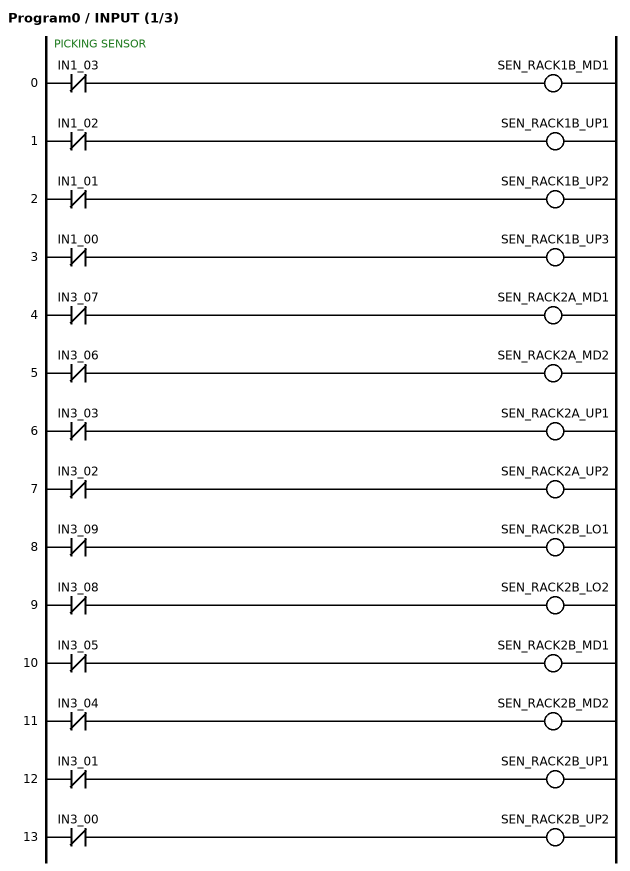
(* [picture p24: Program0 / INPUT, rungs 0-13] *)
(* Rung 0: PICKING SENSOR *)
SEN_RACK1B_MD1 := NOT IN1_03;
(* Rung 1 *)
SEN_RACK1B_UP1 := NOT IN1_02;
(* Rung 2 *)
SEN_RACK1B_UP2 := NOT IN1_01;
(* Rung 3 *)
SEN_RACK1B_UP3 := NOT IN1_00;
(* Rung 4 *)
SEN_RACK2A_MD1 := NOT IN3_07;
(* Rung 5 *)
SEN_RACK2A_MD2 := NOT IN3_06;
(* Rung 6 *)
SEN_RACK2A_UP1 := NOT IN3_03;
(* Rung 7 *)
SEN_RACK2A_UP2 := NOT IN3_02;
(* Rung 8 *)
SEN_RACK2B_LO1 := NOT IN3_09;
(* Rung 9 *)
SEN_RACK2B_LO2 := NOT IN3_08;
(* Rung 10 *)
SEN_RACK2B_MD1 := NOT IN3_05;
(* Rung 11 *)
SEN_RACK2B_MD2 := NOT IN3_04;
(* Rung 12 *)
SEN_RACK2B_UP1 := NOT IN3_01;
(* Rung 13 *)
SEN_RACK2B_UP2 := NOT IN3_00;

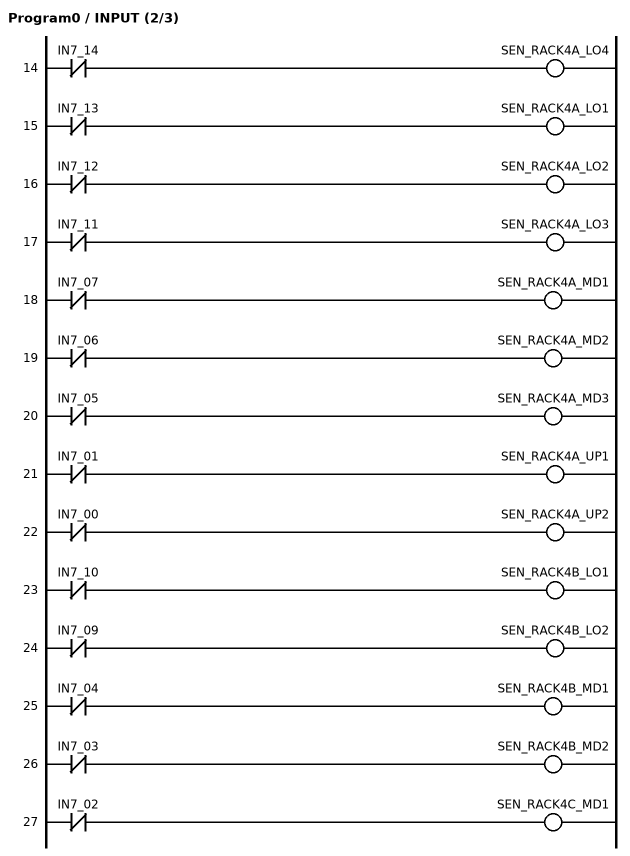
(* Rung 14 *)
SEN_RACK4A_LO4 := NOT IN7_14;
(* Rung 15 *)
SEN_RACK4A_LO1 := NOT IN7_13;
(* Rung 16 *)
SEN_RACK4A_LO2 := NOT IN7_12;
(* Rung 17 *)
SEN_RACK4A_LO3 := NOT IN7_11;
(* Rung 18 *)
SEN_RACK4A_MD1 := NOT IN7_07;
(* Rung 19 *)
SEN_RACK4A_MD2 := NOT IN7_06;
(* Rung 20 *)
SEN_RACK4A_MD3 := NOT IN7_05;
(* Rung 21 *)
SEN_RACK4A_UP1 := NOT IN7_01;
(* Rung 22 *)
SEN_RACK4A_UP2 := NOT IN7_00;
(* Rung 23 *)
SEN_RACK4B_LO1 := NOT IN7_10;
(* Rung 24 *)
SEN_RACK4B_LO2 := NOT IN7_09;
(* Rung 25 *)
SEN_RACK4B_MD1 := NOT IN7_04;
(* Rung 26 *)
SEN_RACK4B_MD2 := NOT IN7_03;
(* Rung 27 *)
SEN_RACK4C_MD1 := NOT IN7_02;

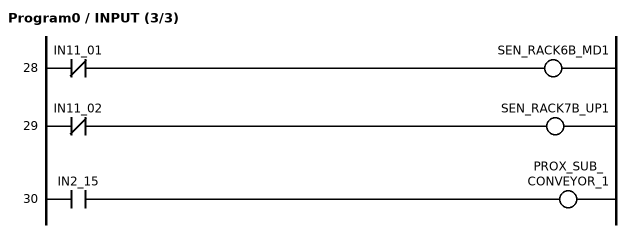
(* Rung 28 *)
SEN_RACK6B_MD1 := NOT IN11_01;
(* Rung 29 *)
SEN_RACK7B_UP1 := NOT IN11_02;
(* Rung 30 *)
PROX_SUB_CONVEYOR_1 := IN2_15;

(* Section OUTPUT: ladder, written here as Structured Text *)

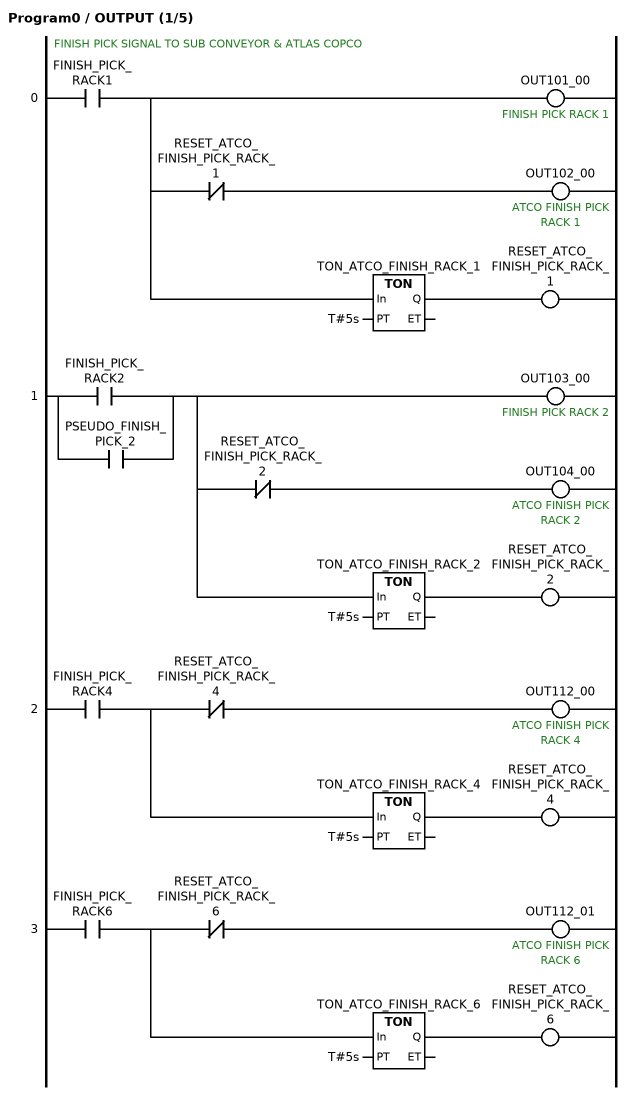
(* Rung 0: FINISH PICK SIGNAL TO SUB CONVEYOR & ATLAS COPCO *)
OUT101_00 := FINISH_PICK_RACK1;
OUT102_00 := FINISH_PICK_RACK1 AND NOT RESET_ATCO_FINISH_PICK_RACK_1;
TON_ATCO_FINISH_RACK_1(In := FINISH_PICK_RACK1, PT := T#5s);
RESET_ATCO_FINISH_PICK_RACK_1 := TON_ATCO_FINISH_RACK_1.Q;
(* Rung 1 *)
OUT103_00 := FINISH_PICK_RACK2 OR PSEUDO_FINISH_PICK_2;
OUT104_00 := (FINISH_PICK_RACK2 OR PSEUDO_FINISH_PICK_2) AND NOT RESET_ATCO_FINISH_PICK_RACK_2;
TON_ATCO_FINISH_RACK_2(In := FINISH_PICK_RACK2 OR PSEUDO_FINISH_PICK_2, PT := T#5s);
RESET_ATCO_FINISH_PICK_RACK_2 := TON_ATCO_FINISH_RACK_2.Q;
(* Rung 2 *)
OUT112_00 := FINISH_PICK_RACK4 AND NOT RESET_ATCO_FINISH_PICK_RACK_4;
TON_ATCO_FINISH_RACK_4(In := FINISH_PICK_RACK4, PT := T#5s);
RESET_ATCO_FINISH_PICK_RACK_4 := TON_ATCO_FINISH_RACK_4.Q;
(* Rung 3 *)
OUT112_01 := FINISH_PICK_RACK6 AND NOT RESET_ATCO_FINISH_PICK_RACK_6;
TON_ATCO_FINISH_RACK_6(In := FINISH_PICK_RACK6, PT := T#5s);
RESET_ATCO_FINISH_PICK_RACK_6 := TON_ATCO_FINISH_RACK_6.Q;

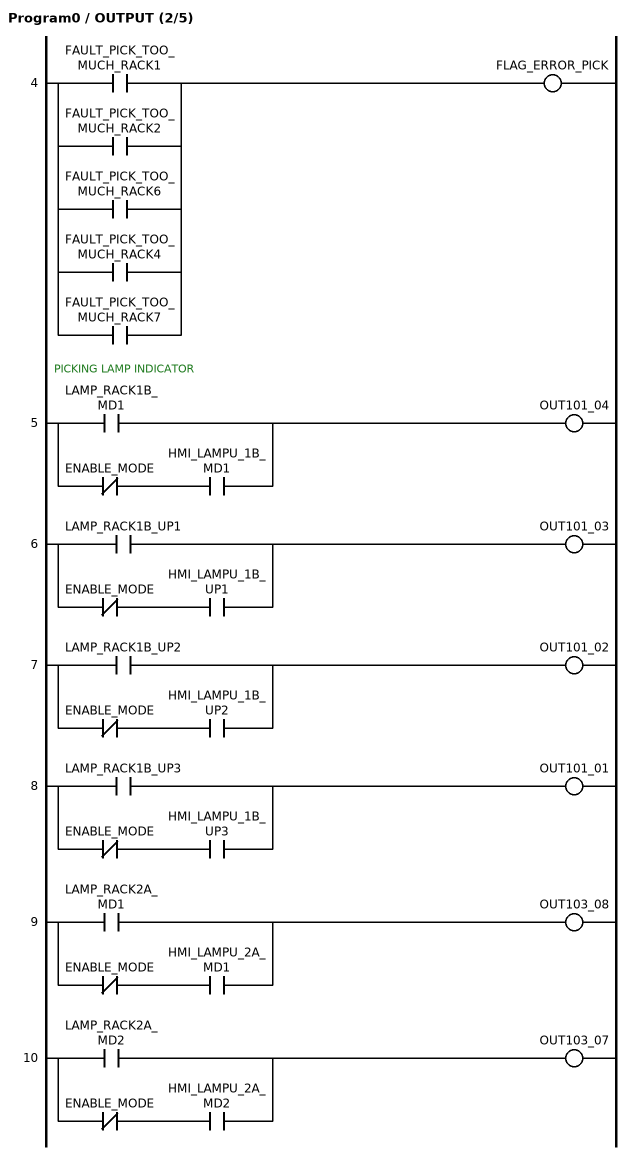
(* Rung 4 *)
FLAG_ERROR_PICK := FAULT_PICK_TOO_MUCH_RACK1 OR FAULT_PICK_TOO_MUCH_RACK2 OR FAULT_PICK_TOO_MUCH_RACK6 OR FAULT_PICK_TOO_MUCH_RACK4 OR FAULT_PICK_TOO_MUCH_RACK7;
(* Rung 5: PICKING LAMP INDICATOR *)
OUT101_04 := LAMP_RACK1B_MD1 OR (NOT ENABLE_MODE AND HMI_LAMPU_1B_MD1);
(* Rung 6 *)
OUT101_03 := LAMP_RACK1B_UP1 OR (NOT ENABLE_MODE AND HMI_LAMPU_1B_UP1);
(* Rung 7 *)
OUT101_02 := LAMP_RACK1B_UP2 OR (NOT ENABLE_MODE AND HMI_LAMPU_1B_UP2);
(* Rung 8 *)
OUT101_01 := LAMP_RACK1B_UP3 OR (NOT ENABLE_MODE AND HMI_LAMPU_1B_UP3);
(* Rung 9 *)
OUT103_08 := LAMP_RACK2A_MD1 OR (NOT ENABLE_MODE AND HMI_LAMPU_2A_MD1);
(* Rung 10 *)
OUT103_07 := LAMP_RACK2A_MD2 OR (NOT ENABLE_MODE AND HMI_LAMPU_2A_MD2);

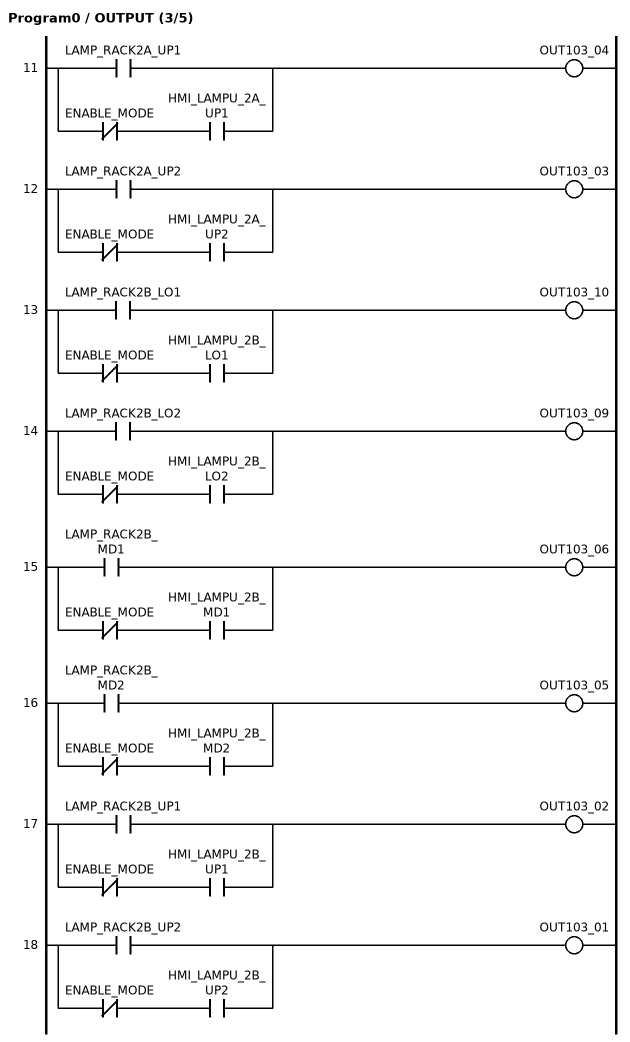
(* Rung 11 *)
OUT103_04 := LAMP_RACK2A_UP1 OR (NOT ENABLE_MODE AND HMI_LAMPU_2A_UP1);
(* Rung 12 *)
OUT103_03 := LAMP_RACK2A_UP2 OR (NOT ENABLE_MODE AND HMI_LAMPU_2A_UP2);
(* Rung 13 *)
OUT103_10 := LAMP_RACK2B_LO1 OR (NOT ENABLE_MODE AND HMI_LAMPU_2B_LO1);
(* Rung 14 *)
OUT103_09 := LAMP_RACK2B_LO2 OR (NOT ENABLE_MODE AND HMI_LAMPU_2B_LO2);
(* Rung 15 *)
OUT103_06 := LAMP_RACK2B_MD1 OR (NOT ENABLE_MODE AND HMI_LAMPU_2B_MD1);
(* Rung 16 *)
OUT103_05 := LAMP_RACK2B_MD2 OR (NOT ENABLE_MODE AND HMI_LAMPU_2B_MD2);
(* Rung 17 *)
OUT103_02 := LAMP_RACK2B_UP1 OR (NOT ENABLE_MODE AND HMI_LAMPU_2B_UP1);
(* Rung 18 *)
OUT103_01 := LAMP_RACK2B_UP2 OR (NOT ENABLE_MODE AND HMI_LAMPU_2B_UP2);

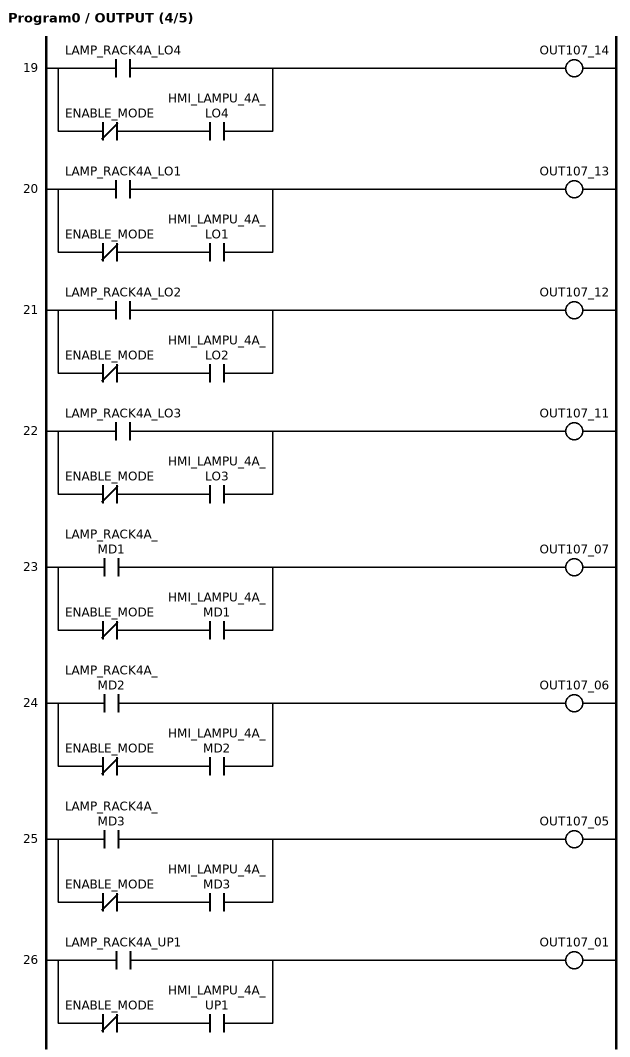
(* Rung 19 *)
OUT107_14 := LAMP_RACK4A_LO4 OR (NOT ENABLE_MODE AND HMI_LAMPU_4A_LO4);
(* Rung 20 *)
OUT107_13 := LAMP_RACK4A_LO1 OR (NOT ENABLE_MODE AND HMI_LAMPU_4A_LO1);
(* Rung 21 *)
OUT107_12 := LAMP_RACK4A_LO2 OR (NOT ENABLE_MODE AND HMI_LAMPU_4A_LO2);
(* Rung 22 *)
OUT107_11 := LAMP_RACK4A_LO3 OR (NOT ENABLE_MODE AND HMI_LAMPU_4A_LO3);
(* Rung 23 *)
OUT107_07 := LAMP_RACK4A_MD1 OR (NOT ENABLE_MODE AND HMI_LAMPU_4A_MD1);
(* Rung 24 *)
OUT107_06 := LAMP_RACK4A_MD2 OR (NOT ENABLE_MODE AND HMI_LAMPU_4A_MD2);
(* Rung 25 *)
OUT107_05 := LAMP_RACK4A_MD3 OR (NOT ENABLE_MODE AND HMI_LAMPU_4A_MD3);
(* Rung 26 *)
OUT107_01 := LAMP_RACK4A_UP1 OR (NOT ENABLE_MODE AND HMI_LAMPU_4A_UP1);

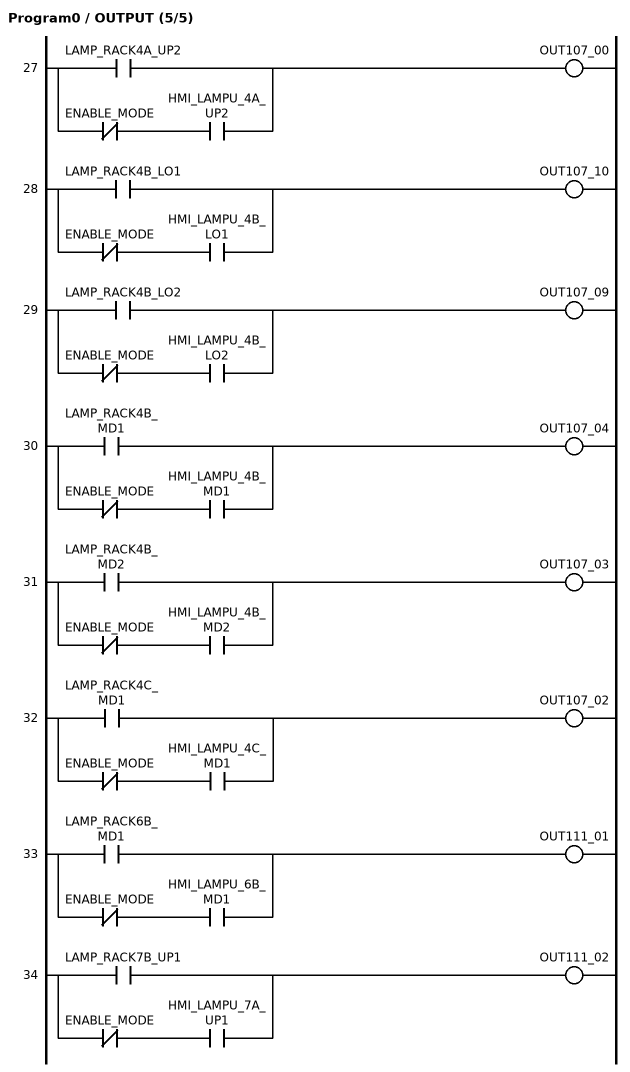
(* Rung 27 *)
OUT107_00 := LAMP_RACK4A_UP2 OR (NOT ENABLE_MODE AND HMI_LAMPU_4A_UP2);
(* Rung 28 *)
OUT107_10 := LAMP_RACK4B_LO1 OR (NOT ENABLE_MODE AND HMI_LAMPU_4B_LO1);
(* Rung 29 *)
OUT107_09 := LAMP_RACK4B_LO2 OR (NOT ENABLE_MODE AND HMI_LAMPU_4B_LO2);
(* Rung 30 *)
OUT107_04 := LAMP_RACK4B_MD1 OR (NOT ENABLE_MODE AND HMI_LAMPU_4B_MD1);
(* Rung 31 *)
OUT107_03 := LAMP_RACK4B_MD2 OR (NOT ENABLE_MODE AND HMI_LAMPU_4B_MD2);
(* Rung 32 *)
OUT107_02 := LAMP_RACK4C_MD1 OR (NOT ENABLE_MODE AND HMI_LAMPU_4C_MD1);
(* Rung 33 *)
OUT111_01 := LAMP_RACK6B_MD1 OR (NOT ENABLE_MODE AND HMI_LAMPU_6B_MD1);
(* Rung 34 *)
OUT111_02 := LAMP_RACK7B_UP1 OR (NOT ENABLE_MODE AND HMI_LAMPU_7A_UP1);
END_PROGRAM

FUNCTION_BLOCK FB_PICKING_SEQ
VAR
    DONE_PICK_1 : BOOL;
    NI_LAMP_PICK_1 : BOOL;
    NI_FAULT_MUCH_LAMP_PICK_1 : BOOL;
    NI_FAULT_FALSE_LAMP_PICK_1 : BOOL;
    DONE_PICK_2 : BOOL;
    NI_LAMP_PICK_2 : BOOL;
    NI_FAULT_MUCH_LAMP_PICK_2 : BOOL;
    NI_FAULT_FALSE_LAMP_PICK_2 : BOOL;
    DONE_PICK_3 : BOOL;
    NI_LAMP_PICK_3 : BOOL;
    NI_FAULT_MUCH_LAMP_PICK_3 : BOOL;
    NI_FAULT_FALSE_LAMP_PICK_3 : BOOL;
    DONE_PICK_4 : BOOL;
    NI_LAMP_PICK_4 : BOOL;
    NI_FAULT_MUCH_LAMP_PICK_4 : BOOL;
    NI_FAULT_FALSE_LAMP_PICK_4 : BOOL;
    DONE_PICK_5 : BOOL;
    NI_LAMP_PICK_5 : BOOL;
    NI_FAULT_MUCH_LAMP_PICK_5 : BOOL;
    NI_FAULT_FALSE_LAMP_PICK_5 : BOOL;
    DONE_PICK_6 : BOOL;
    NI_LAMP_PICK_6 : BOOL;
    NI_FAULT_MUCH_LAMP_PICK_6 : BOOL;
    NI_FAULT_FALSE_LAMP_PICK_6 : BOOL;
    DONE_PICK_7 : BOOL;
    NI_LAMP_PICK_7 : BOOL;
    NI_FAULT_MUCH_LAMP_PICK_7 : BOOL;
    NI_FAULT_FALSE_LAMP_PICK_7 : BOOL;
    NI_LAMP_PICK_8 : BOOL;
    DONE_PICK_8 : BOOL;
    NI_FAULT_MUCH_LAMP_PICK_8 : BOOL;
    NI_FAULT_FALSE_LAMP_PICK_8 : BOOL;
    DONE_PICK_9 : BOOL;
    NI_LAMP_PICK_9 : BOOL;
    NI_FAULT_MUCH_LAMP_PICK_9 : BOOL;
    NI_FAULT_FALSE_LAMP_PICK_9 : BOOL;
    DONE_PICK_10 : BOOL;
    NI_LAMP_PICK_10 : BOOL;
    NI_FAULT_MUCH_LAMP_PICK_10 : BOOL;
    NI_FAULT_FALSE_LAMP_PICK_10 : BOOL;
    NI_LAMP_PICK_11 : BOOL;
    DONE_PICK_11 : BOOL;
    NI_FAULT_MUCH_LAMP_PICK_11 : BOOL;
    NI_FAULT_FALSE_LAMP_PICK_11 : BOOL;
    DONE_PICK_12 : BOOL;
    NI_LAMP_PICK_12 : BOOL;
    NI_FAULT_MUCH_LAMP_PICK_12 : BOOL;
    NI_FAULT_FALSE_LAMP_PICK_12 : BOOL;
    DONE_PICK_13 : BOOL;
    NI_LAMP_PICK_13 : BOOL;
    NI_FAULT_MUCH_LAMP_PICK_13 : BOOL;
    NI_FAULT_FALSE_LAMP_PICK_14 : BOOL;
    NI_LAMP_PICK_14 : BOOL;
    NI_FAULT_FALSE_LAMP_PICK_13 : BOOL;
    DONE_PICK_14 : BOOL;
    NI_FAULT_MUCH_LAMP_PICK_14 : BOOL;
    DONE_PICK_15 : BOOL;
    NI_LAMP_PICK_15 : BOOL;
    NI_FAULT_MUCH_LAMP_PICK_15 : BOOL;
    NI_FAULT_FALSE_LAMP_PICK_15 : BOOL;
    NI_LAMP_PICK_16 : BOOL;
    DONE_PICK_16 : BOOL;
    NI_FAULT_MUCH_LAMP_PICK_16 : BOOL;
    NI_FAULT_FALSE_LAMP_PICK_16 : BOOL;
    DONE_PICK_17 : BOOL;
    NI_LAMP_PICK_17 : BOOL;
    NI_FAULT_MUCH_LAMP_PICK_17 : BOOL;
    NI_FAULT_FALSE_LAMP_PICK_17 : BOOL;
    DONE_PICK_18 : BOOL;
    NI_LAMP_PICK_18 : BOOL;
    NI_FAULT_MUCH_LAMP_PICK_18 : BOOL;
    NI_FAULT_FALSE_LAMP_PICK_18 : BOOL;
    NI_LAMP_PICK_19 : BOOL;
    DONE_PICK_19 : BOOL;
    NI_FAULT_MUCH_LAMP_PICK_19 : BOOL;
    NI_FAULT_FALSE_LAMP_PICK_19 : BOOL;
    DONE_PICK_20 : BOOL;
    NI_LAMP_PICK_20 : BOOL;
    NI_FAULT_MUCH_LAMP_PICK_20 : BOOL;
    NI_FAULT_FALSE_LAMP_PICK_20 : BOOL;
    ALL_NI_LAMP_PICK : BOOL;
    ALL_LI_LAMP_PICK : BOOL;
    ALL_NI_FAULT_FALSE_LAMP_PICK : BOOL;
    ALL_LI_FAULT_FALSE_LAMP_PICK : BOOL;
    ALL_NI_FAULT_TOO_MUCH_LAMP_PICK : BOOL;
    ALL_LI_FAULT_TOO_MUCH_LAMP_PICK : BOOL;
    AFTER_PICK_1 : BOOL;
    TON_AFTER_PICK_1 : TON;
    LI_LAMP_PICK_1 : BOOL;
    AFTER_PICK_2 : BOOL;
    LI_LAMP_PICK_2 : BOOL;
    TON_AFTER_PICK_2 : TON;
    AFTER_PICK_3 : BOOL;
    LI_LAMP_PICK_3 : BOOL;
    TON_AFTER_PICK_3 : TON;
    LI_LAMP_PICK_4 : BOOL;
    AFTER_PICK_4 : BOOL;
    TON_AFTER_PICK_4 : TON;
    AFTER_PICK_5 : BOOL;
    LI_LAMP_PICK_5 : BOOL;
    TON_AFTER_PICK_5 : TON;
    AFTER_PICK_6 : BOOL;
    LI_LAMP_PICK_6 : BOOL;
    TON_AFTER_PICK_6 : TON;
    LI_LAMP_PICK_7 : BOOL;
    AFTER_PICK_7 : BOOL;
    TON_AFTER_PICK_7 : TON;
    AFTER_PICK_8 : BOOL;
    LI_LAMP_PICK_8 : BOOL;
    TON_AFTER_PICK_8 : TON;
    AFTER_PICK_9 : BOOL;
    LI_LAMP_PICK_9 : BOOL;
    TON_AFTER_PICK_9 : TON;
    LI_LAMP_PICK_10 : BOOL;
    AFTER_PICK_10 : BOOL;
    TON_AFTER_PICK_10 : TON;
    LI_LAMP_PICK_11 : BOOL;
    LI_LAMP_PICK_12 : BOOL;
    LI_LAMP_PICK_13 : BOOL;
    LI_LAMP_PICK_14 : BOOL;
    LI_LAMP_PICK_15 : BOOL;
    LI_LAMP_PICK_16 : BOOL;
    LI_LAMP_PICK_17 : BOOL;
    LI_LAMP_PICK_18 : BOOL;
    LI_LAMP_PICK_19 : BOOL;
    LI_LAMP_PICK_20 : BOOL;
    AFTER_PICK_11 : BOOL;
    TON_AFTER_PICK_11 : TON;
    AFTER_PICK_12 : BOOL;
    TON_AFTER_PICK_12 : TON;
    AFTER_PICK_13 : BOOL;
    TON_AFTER_PICK_13 : TON;
    AFTER_PICK_14 : BOOL;
    TON_AFTER_PICK_14 : TON;
    AFTER_PICK_15 : BOOL;
    TON_AFTER_PICK_15 : TON;
    AFTER_PICK_16 : BOOL;
    TON_AFTER_PICK_16 : TON;
    AFTER_PICK_17 : BOOL;
    TON_AFTER_PICK_17 : TON;
    AFTER_PICK_18 : BOOL;
    TON_AFTER_PICK_18 : TON;
    AFTER_PICK_19 : BOOL;
    TON_AFTER_PICK_19 : TON;
    AFTER_PICK_20 : BOOL;
    TON_AFTER_PICK_20 : TON;
END_VAR
VAR_INPUT
    ENABLE : BOOL;
    NICKEL : BOOL;
    LITHIUM : BOOL;
    SEN_PICK_1 : BOOL;
    SEN_PICK_2 : BOOL;
    SEN_PICK_3 : BOOL;
    SEN_PICK_4 : BOOL;
    SEN_PICK_5 : BOOL;
    SEN_PICK_6 : BOOL;
    SEN_PICK_7 : BOOL;
    SEN_PICK_8 : BOOL;
    SEN_PICK_9 : BOOL;
    SEN_PICK_10 : BOOL;
    SEN_PICK_11 : BOOL;
    SEN_PICK_12 : BOOL;
    SEN_PICK_13 : BOOL;
    SEN_PICK_14 : BOOL;
    SEN_PICK_15 : BOOL;
    SEN_PICK_16 : BOOL;
    SEN_PICK_17 : BOOL;
    SEN_PICK_18 : BOOL;
    SEN_PICK_19 : BOOL;
    SEN_PICK_20 : BOOL;
END_VAR
VAR_OUTPUT
    ENABLE_OUT : BOOL;
    FINISH_PICK : BOOL;
    FAULT_PICK_FALSE : BOOL;
    FAULT_PICK_TOO_MUCH : BOOL;
    LAMP_PICK_1 : BOOL;
    LAMP_PICK_2 : BOOL;
    LAMP_PICK_3 : BOOL;
    LAMP_PICK_4 : BOOL;
    LAMP_PICK_5 : BOOL;
    LAMP_PICK_6 : BOOL;
    LAMP_PICK_7 : BOOL;
    LAMP_PICK_8 : BOOL;
    LAMP_PICK_9 : BOOL;
    LAMP_PICK_10 : BOOL;
    LAMP_PICK_11 : BOOL;
    LAMP_PICK_12 : BOOL;
    LAMP_PICK_13 : BOOL;
    LAMP_PICK_14 : BOOL;
    LAMP_PICK_15 : BOOL;
    LAMP_PICK_16 : BOOL;
    LAMP_PICK_17 : BOOL;
    LAMP_PICK_18 : BOOL;
    LAMP_PICK_19 : BOOL;
    LAMP_PICK_20 : BOOL;
END_VAR
VAR_INPUT
    TEACH_PICK_1 : WORD;
    TEACH_PICK_2 : WORD;
    TEACH_PICK_3 : WORD;
    TEACH_PICK_4 : WORD;
    TEACH_PICK_5 : WORD;
    TEACH_PICK_6 : WORD;
    TEACH_PICK_7 : WORD;
    TEACH_PICK_8 : WORD;
    TEACH_PICK_9 : WORD;
    TEACH_PICK_10 : WORD;
    TEACH_PICK_11 : WORD;
    TEACH_PICK_12 : WORD;
    TEACH_PICK_13 : WORD;
    TEACH_PICK_14 : WORD;
    TEACH_PICK_15 : WORD;
    TEACH_PICK_16 : WORD;
    TEACH_PICK_17 : WORD;
    TEACH_PICK_18 : WORD;
    TEACH_PICK_19 : WORD;
    TEACH_PICK_20 : WORD;
END_VAR
VAR_OUTPUT
    RESET_TIMER_TOO_LONG : BOOL;
END_VAR
VAR
    _p1 : BOOL;
    _p2 : BOOL;
    _p3 : BOOL;
    _p4 : BOOL;
    _p5 : BOOL;
    _p6 : BOOL;
    _p7 : BOOL;
    _p8 : BOOL;
    _p9 : BOOL;
    _p10 : BOOL;
    _p11 : BOOL;
    _e12 : F_TRIG;
    _e13 : F_TRIG;
    _e14 : F_TRIG;
    _e15 : F_TRIG;
    _e16 : F_TRIG;
    _e17 : F_TRIG;
    _e18 : F_TRIG;
    _e19 : F_TRIG;
    _e20 : F_TRIG;
    _e21 : F_TRIG;
    _e22 : F_TRIG;
    _e23 : F_TRIG;
    _e24 : F_TRIG;
    _e25 : F_TRIG;
    _e26 : F_TRIG;
    _e27 : F_TRIG;
    _e28 : F_TRIG;
    _e29 : F_TRIG;
    _e30 : F_TRIG;
    _e31 : F_TRIG;
    _e32 : F_TRIG;
    _e33 : F_TRIG;
    _e34 : F_TRIG;
    _e35 : F_TRIG;
    _e36 : F_TRIG;
    _e37 : F_TRIG;
    _e38 : F_TRIG;
    _e39 : F_TRIG;
    _e40 : F_TRIG;
    _e41 : F_TRIG;
    _e42 : F_TRIG;
    _e43 : F_TRIG;
    _e44 : F_TRIG;
    _e45 : F_TRIG;
    _e46 : F_TRIG;
    _e47 : F_TRIG;
    _e48 : F_TRIG;
    _e49 : F_TRIG;
    _e50 : F_TRIG;
    _e51 : F_TRIG;
    _e52 : F_TRIG;
    _e53 : F_TRIG;
    _e54 : F_TRIG;
    _e55 : F_TRIG;
    _e56 : F_TRIG;
    _e57 : F_TRIG;
    _e58 : F_TRIG;
    _e59 : F_TRIG;
    _e60 : F_TRIG;
    _e61 : F_TRIG;
    _e62 : F_TRIG;
    _e63 : F_TRIG;
    _e64 : F_TRIG;
    _e65 : F_TRIG;
    _e66 : F_TRIG;
    _e67 : F_TRIG;
    _e68 : F_TRIG;
    _e69 : F_TRIG;
    _e70 : F_TRIG;
    _e71 : F_TRIG;
    _e72 : F_TRIG;
    _e73 : F_TRIG;
    _e74 : F_TRIG;
    _e75 : F_TRIG;
    _e76 : F_TRIG;
    _e77 : F_TRIG;
    _e78 : F_TRIG;
    _e79 : F_TRIG;
    _e80 : F_TRIG;
    _e81 : F_TRIG;
    _e82 : F_TRIG;
    _e83 : F_TRIG;
    _e84 : F_TRIG;
    _e85 : F_TRIG;
    _e86 : F_TRIG;
    _e87 : F_TRIG;
    _e88 : F_TRIG;
    _e89 : F_TRIG;
    _e90 : F_TRIG;
    _e91 : F_TRIG;
    _e92 : F_TRIG;
    _e93 : F_TRIG;
    _e94 : F_TRIG;
    _e95 : F_TRIG;
    _e96 : F_TRIG;
    _e97 : F_TRIG;
    _e98 : F_TRIG;
    _e99 : F_TRIG;
    _e100 : F_TRIG;
    _e101 : F_TRIG;
    _e102 : F_TRIG;
    _e103 : F_TRIG;
    _e104 : F_TRIG;
    _e105 : F_TRIG;
    _e106 : F_TRIG;
    _e107 : F_TRIG;
    _e108 : F_TRIG;
    _e109 : F_TRIG;
    _e110 : F_TRIG;
    _e111 : F_TRIG;
    _e112 : F_TRIG;
    _e113 : F_TRIG;
    _e114 : F_TRIG;
    _e115 : F_TRIG;
    _e116 : F_TRIG;
    _e117 : F_TRIG;
    _e118 : F_TRIG;
    _e119 : F_TRIG;
    _e120 : F_TRIG;
    _e121 : F_TRIG;
    _e122 : F_TRIG;
    _e123 : F_TRIG;
    _e124 : F_TRIG;
    _e125 : F_TRIG;
    _e126 : F_TRIG;
    _e127 : F_TRIG;
    _e128 : F_TRIG;
    _e129 : F_TRIG;
    _e130 : F_TRIG;
    _e131 : F_TRIG;
END_VAR
(* ladder, written here as Structured Text *)

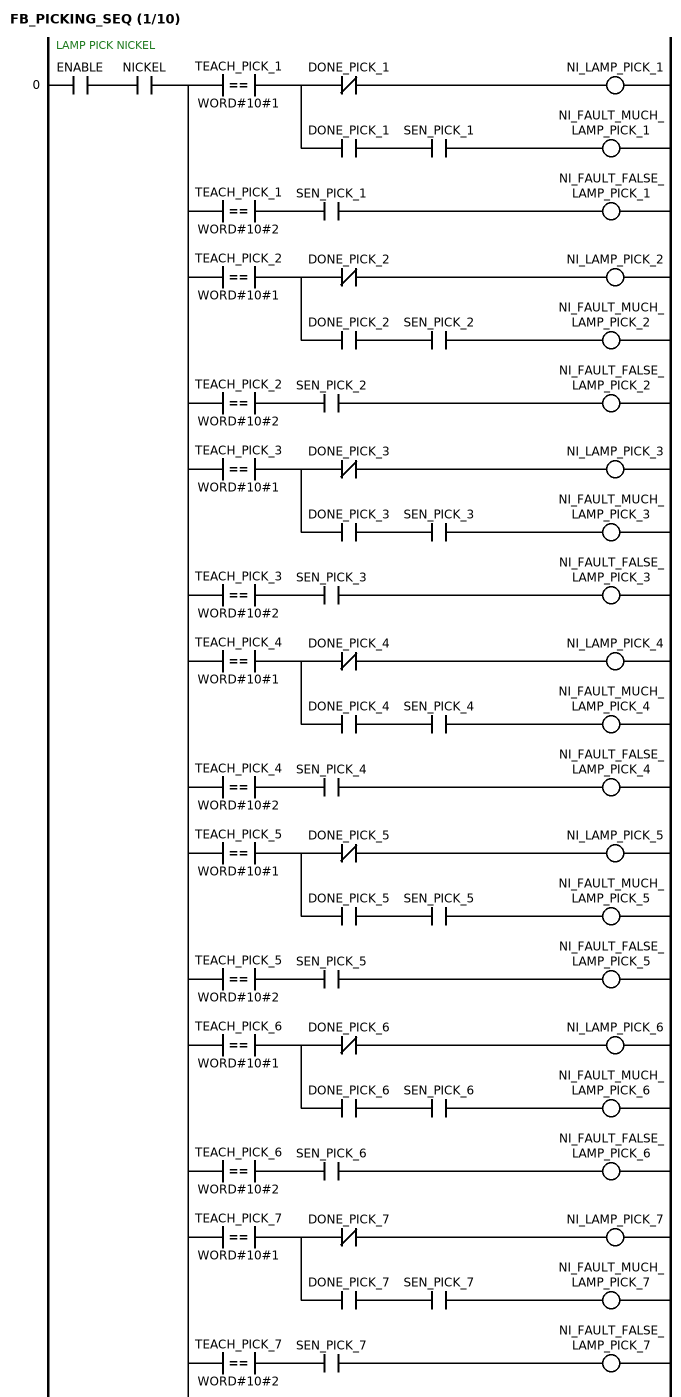

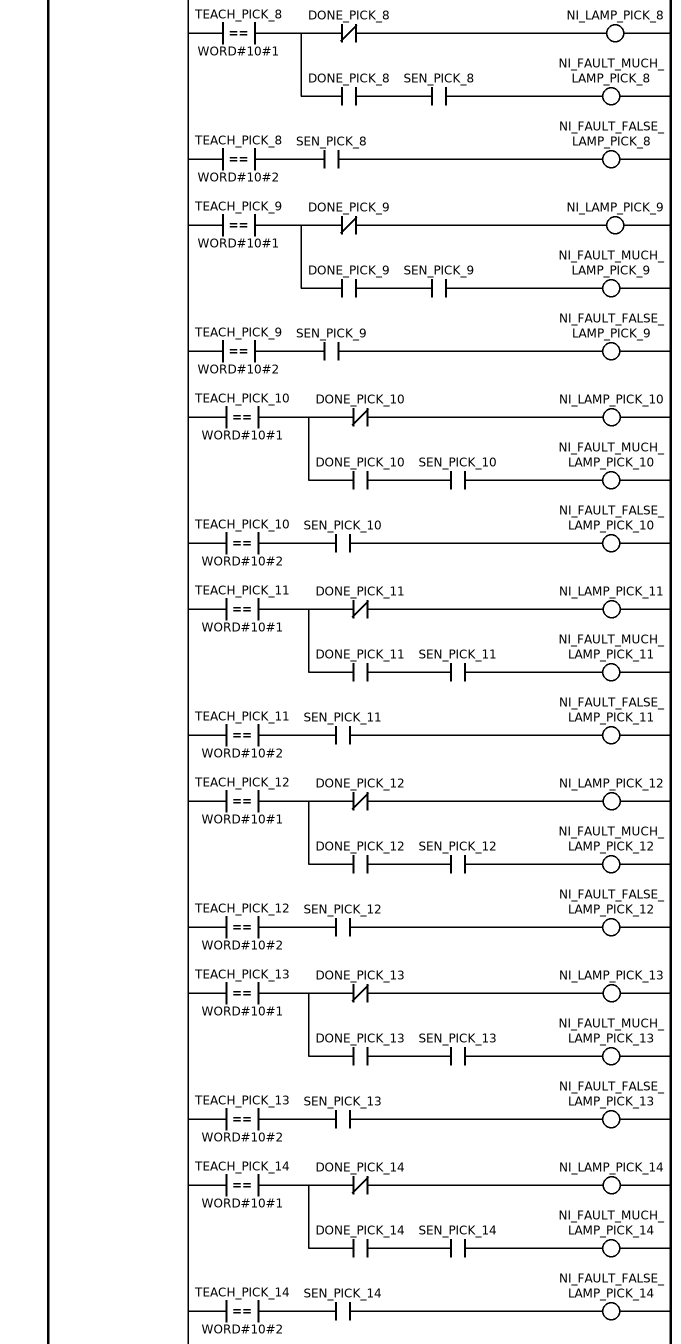

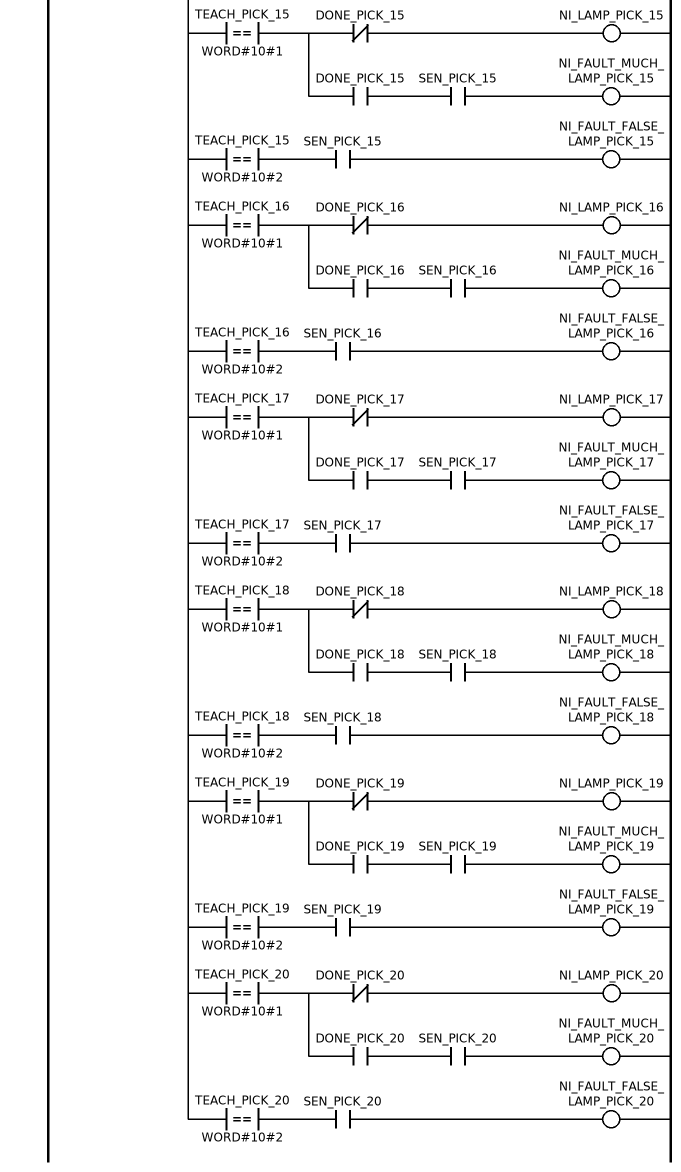
(* Rung 0: LAMP PICK NICKEL *)
NI_LAMP_PICK_1 := ENABLE AND NICKEL AND (TEACH_PICK_1 = WORD#10#1) AND NOT DONE_PICK_1;
NI_FAULT_MUCH_LAMP_PICK_1 := ENABLE AND NICKEL AND (TEACH_PICK_1 = WORD#10#1) AND DONE_PICK_1 AND SEN_PICK_1;
NI_FAULT_FALSE_LAMP_PICK_1 := ENABLE AND NICKEL AND (TEACH_PICK_1 = WORD#10#2) AND SEN_PICK_1;
NI_LAMP_PICK_2 := ENABLE AND NICKEL AND (TEACH_PICK_2 = WORD#10#1) AND NOT DONE_PICK_2;
NI_FAULT_MUCH_LAMP_PICK_2 := ENABLE AND NICKEL AND (TEACH_PICK_2 = WORD#10#1) AND DONE_PICK_2 AND SEN_PICK_2;
NI_FAULT_FALSE_LAMP_PICK_2 := ENABLE AND NICKEL AND (TEACH_PICK_2 = WORD#10#2) AND SEN_PICK_2;
NI_LAMP_PICK_3 := ENABLE AND NICKEL AND (TEACH_PICK_3 = WORD#10#1) AND NOT DONE_PICK_3;
NI_FAULT_MUCH_LAMP_PICK_3 := ENABLE AND NICKEL AND (TEACH_PICK_3 = WORD#10#1) AND DONE_PICK_3 AND SEN_PICK_3;
NI_FAULT_FALSE_LAMP_PICK_3 := ENABLE AND NICKEL AND (TEACH_PICK_3 = WORD#10#2) AND SEN_PICK_3;
NI_LAMP_PICK_4 := ENABLE AND NICKEL AND (TEACH_PICK_4 = WORD#10#1) AND NOT DONE_PICK_4;
NI_FAULT_MUCH_LAMP_PICK_4 := ENABLE AND NICKEL AND (TEACH_PICK_4 = WORD#10#1) AND DONE_PICK_4 AND SEN_PICK_4;
NI_FAULT_FALSE_LAMP_PICK_4 := ENABLE AND NICKEL AND (TEACH_PICK_4 = WORD#10#2) AND SEN_PICK_4;
NI_LAMP_PICK_5 := ENABLE AND NICKEL AND (TEACH_PICK_5 = WORD#10#1) AND NOT DONE_PICK_5;
NI_FAULT_MUCH_LAMP_PICK_5 := ENABLE AND NICKEL AND (TEACH_PICK_5 = WORD#10#1) AND DONE_PICK_5 AND SEN_PICK_5;
NI_FAULT_FALSE_LAMP_PICK_5 := ENABLE AND NICKEL AND (TEACH_PICK_5 = WORD#10#2) AND SEN_PICK_5;
NI_LAMP_PICK_6 := ENABLE AND NICKEL AND (TEACH_PICK_6 = WORD#10#1) AND NOT DONE_PICK_6;
NI_FAULT_MUCH_LAMP_PICK_6 := ENABLE AND NICKEL AND (TEACH_PICK_6 = WORD#10#1) AND DONE_PICK_6 AND SEN_PICK_6;
NI_FAULT_FALSE_LAMP_PICK_6 := ENABLE AND NICKEL AND (TEACH_PICK_6 = WORD#10#2) AND SEN_PICK_6;
NI_LAMP_PICK_7 := ENABLE AND NICKEL AND (TEACH_PICK_7 = WORD#10#1) AND NOT DONE_PICK_7;
NI_FAULT_MUCH_LAMP_PICK_7 := ENABLE AND NICKEL AND (TEACH_PICK_7 = WORD#10#1) AND DONE_PICK_7 AND SEN_PICK_7;
NI_FAULT_FALSE_LAMP_PICK_7 := ENABLE AND NICKEL AND (TEACH_PICK_7 = WORD#10#2) AND SEN_PICK_7;
NI_LAMP_PICK_8 := ENABLE AND NICKEL AND (TEACH_PICK_8 = WORD#10#1) AND NOT DONE_PICK_8;
NI_FAULT_MUCH_LAMP_PICK_8 := ENABLE AND NICKEL AND (TEACH_PICK_8 = WORD#10#1) AND DONE_PICK_8 AND SEN_PICK_8;
NI_FAULT_FALSE_LAMP_PICK_8 := ENABLE AND NICKEL AND (TEACH_PICK_8 = WORD#10#2) AND SEN_PICK_8;
NI_LAMP_PICK_9 := ENABLE AND NICKEL AND (TEACH_PICK_9 = WORD#10#1) AND NOT DONE_PICK_9;
NI_FAULT_MUCH_LAMP_PICK_9 := ENABLE AND NICKEL AND (TEACH_PICK_9 = WORD#10#1) AND DONE_PICK_9 AND SEN_PICK_9;
NI_FAULT_FALSE_LAMP_PICK_9 := ENABLE AND NICKEL AND (TEACH_PICK_9 = WORD#10#2) AND SEN_PICK_9;
_p1 := ENABLE AND NICKEL AND (TEACH_PICK_10 = WORD#10#1);
NI_LAMP_PICK_10 := _p1 AND NOT DONE_PICK_10;
NI_FAULT_MUCH_LAMP_PICK_10 := _p1 AND DONE_PICK_10 AND SEN_PICK_10;
NI_FAULT_FALSE_LAMP_PICK_10 := ENABLE AND NICKEL AND (TEACH_PICK_10 = WORD#10#2) AND SEN_PICK_10;
_p2 := ENABLE AND NICKEL AND (TEACH_PICK_11 = WORD#10#1);
NI_LAMP_PICK_11 := _p2 AND NOT DONE_PICK_11;
NI_FAULT_MUCH_LAMP_PICK_11 := _p2 AND DONE_PICK_11 AND SEN_PICK_11;
NI_FAULT_FALSE_LAMP_PICK_11 := ENABLE AND NICKEL AND (TEACH_PICK_11 = WORD#10#2) AND SEN_PICK_11;
_p3 := ENABLE AND NICKEL AND (TEACH_PICK_12 = WORD#10#1);
NI_LAMP_PICK_12 := _p3 AND NOT DONE_PICK_12;
NI_FAULT_MUCH_LAMP_PICK_12 := _p3 AND DONE_PICK_12 AND SEN_PICK_12;
NI_FAULT_FALSE_LAMP_PICK_12 := ENABLE AND NICKEL AND (TEACH_PICK_12 = WORD#10#2) AND SEN_PICK_12;
_p4 := ENABLE AND NICKEL AND (TEACH_PICK_13 = WORD#10#1);
NI_LAMP_PICK_13 := _p4 AND NOT DONE_PICK_13;
NI_FAULT_MUCH_LAMP_PICK_13 := _p4 AND DONE_PICK_13 AND SEN_PICK_13;
NI_FAULT_FALSE_LAMP_PICK_13 := ENABLE AND NICKEL AND (TEACH_PICK_13 = WORD#10#2) AND SEN_PICK_13;
_p5 := ENABLE AND NICKEL AND (TEACH_PICK_14 = WORD#10#1);
NI_LAMP_PICK_14 := _p5 AND NOT DONE_PICK_14;
NI_FAULT_MUCH_LAMP_PICK_14 := _p5 AND DONE_PICK_14 AND SEN_PICK_14;
NI_FAULT_FALSE_LAMP_PICK_14 := ENABLE AND NICKEL AND (TEACH_PICK_14 = WORD#10#2) AND SEN_PICK_14;
_p6 := ENABLE AND NICKEL AND (TEACH_PICK_15 = WORD#10#1);
NI_LAMP_PICK_15 := _p6 AND NOT DONE_PICK_15;
NI_FAULT_MUCH_LAMP_PICK_15 := _p6 AND DONE_PICK_15 AND SEN_PICK_15;
NI_FAULT_FALSE_LAMP_PICK_15 := ENABLE AND NICKEL AND (TEACH_PICK_15 = WORD#10#2) AND SEN_PICK_15;
_p7 := ENABLE AND NICKEL AND (TEACH_PICK_16 = WORD#10#1);
NI_LAMP_PICK_16 := _p7 AND NOT DONE_PICK_16;
NI_FAULT_MUCH_LAMP_PICK_16 := _p7 AND DONE_PICK_16 AND SEN_PICK_16;
NI_FAULT_FALSE_LAMP_PICK_16 := ENABLE AND NICKEL AND (TEACH_PICK_16 = WORD#10#2) AND SEN_PICK_16;
_p8 := ENABLE AND NICKEL AND (TEACH_PICK_17 = WORD#10#1);
NI_LAMP_PICK_17 := _p8 AND NOT DONE_PICK_17;
NI_FAULT_MUCH_LAMP_PICK_17 := _p8 AND DONE_PICK_17 AND SEN_PICK_17;
NI_FAULT_FALSE_LAMP_PICK_17 := ENABLE AND NICKEL AND (TEACH_PICK_17 = WORD#10#2) AND SEN_PICK_17;
_p9 := ENABLE AND NICKEL AND (TEACH_PICK_18 = WORD#10#1);
NI_LAMP_PICK_18 := _p9 AND NOT DONE_PICK_18;
NI_FAULT_MUCH_LAMP_PICK_18 := _p9 AND DONE_PICK_18 AND SEN_PICK_18;
NI_FAULT_FALSE_LAMP_PICK_18 := ENABLE AND NICKEL AND (TEACH_PICK_18 = WORD#10#2) AND SEN_PICK_18;
_p10 := ENABLE AND NICKEL AND (TEACH_PICK_19 = WORD#10#1);
NI_LAMP_PICK_19 := _p10 AND NOT DONE_PICK_19;
NI_FAULT_MUCH_LAMP_PICK_19 := _p10 AND DONE_PICK_19 AND SEN_PICK_19;
NI_FAULT_FALSE_LAMP_PICK_19 := ENABLE AND NICKEL AND (TEACH_PICK_19 = WORD#10#2) AND SEN_PICK_19;
_p11 := ENABLE AND NICKEL AND (TEACH_PICK_20 = WORD#10#1);
NI_LAMP_PICK_20 := _p11 AND NOT DONE_PICK_20;
NI_FAULT_MUCH_LAMP_PICK_20 := _p11 AND DONE_PICK_20 AND SEN_PICK_20;
NI_FAULT_FALSE_LAMP_PICK_20 := ENABLE AND NICKEL AND (TEACH_PICK_20 = WORD#10#2) AND SEN_PICK_20;

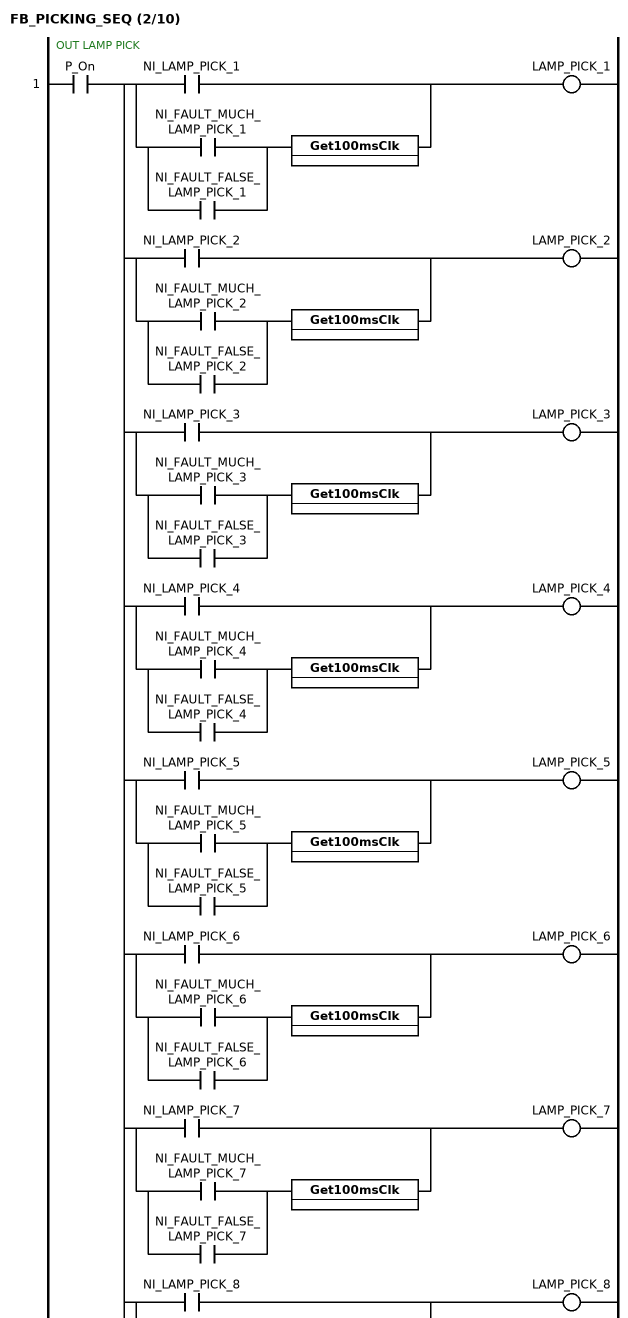

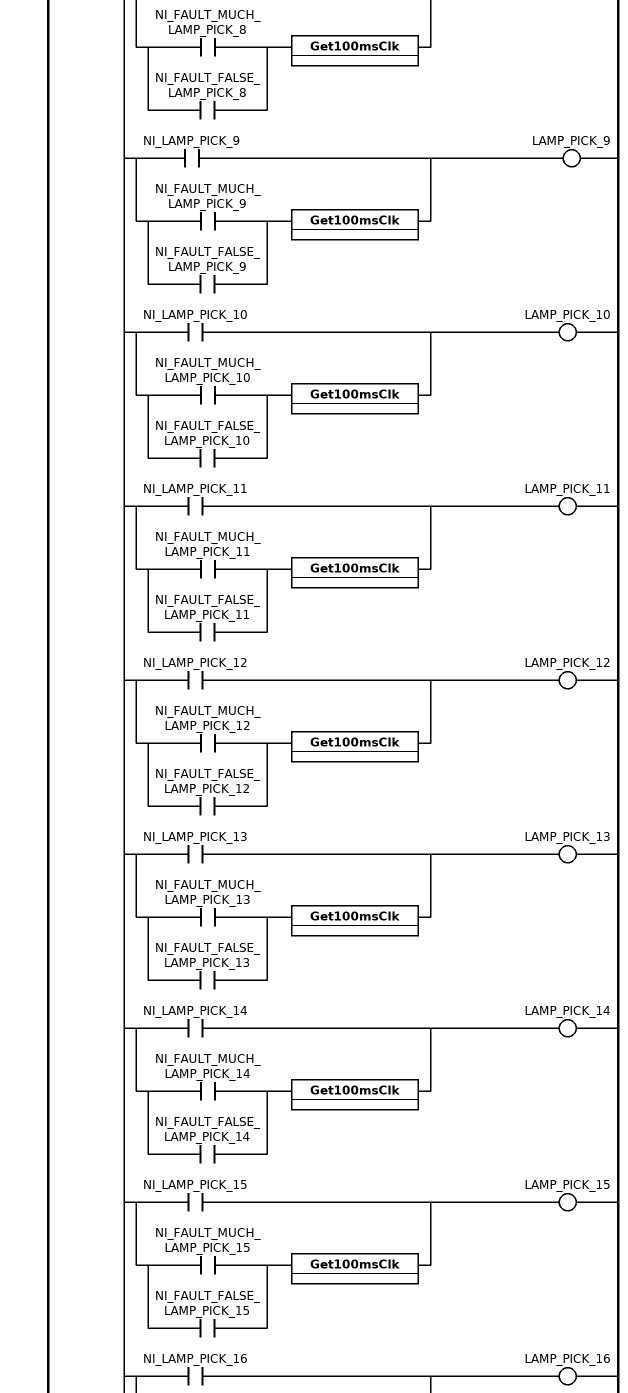

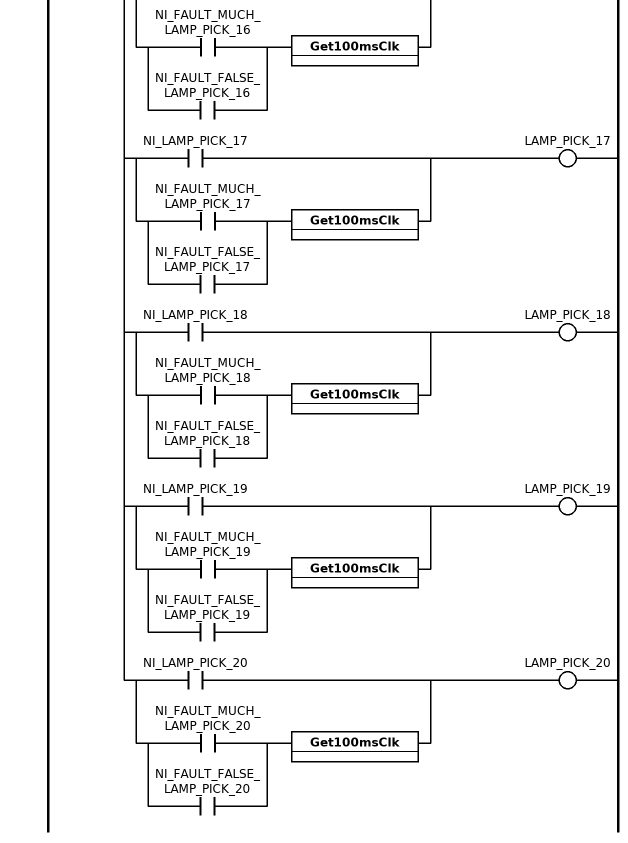
(* Rung 1: OUT LAMP PICK *)
LAMP_PICK_1 := P_On AND (NI_LAMP_PICK_1 OR ((NI_FAULT_MUCH_LAMP_PICK_1 OR NI_FAULT_FALSE_LAMP_PICK_1) AND Get100msClk()));
LAMP_PICK_2 := P_On AND (NI_LAMP_PICK_2 OR ((NI_FAULT_MUCH_LAMP_PICK_2 OR NI_FAULT_FALSE_LAMP_PICK_2) AND Get100msClk()));
LAMP_PICK_3 := P_On AND (NI_LAMP_PICK_3 OR ((NI_FAULT_MUCH_LAMP_PICK_3 OR NI_FAULT_FALSE_LAMP_PICK_3) AND Get100msClk()));
LAMP_PICK_4 := P_On AND (NI_LAMP_PICK_4 OR ((NI_FAULT_MUCH_LAMP_PICK_4 OR NI_FAULT_FALSE_LAMP_PICK_4) AND Get100msClk()));
LAMP_PICK_5 := P_On AND (NI_LAMP_PICK_5 OR ((NI_FAULT_MUCH_LAMP_PICK_5 OR NI_FAULT_FALSE_LAMP_PICK_5) AND Get100msClk()));
LAMP_PICK_6 := P_On AND (NI_LAMP_PICK_6 OR ((NI_FAULT_MUCH_LAMP_PICK_6 OR NI_FAULT_FALSE_LAMP_PICK_6) AND Get100msClk()));
LAMP_PICK_7 := P_On AND (NI_LAMP_PICK_7 OR ((NI_FAULT_MUCH_LAMP_PICK_7 OR NI_FAULT_FALSE_LAMP_PICK_7) AND Get100msClk()));
LAMP_PICK_8 := P_On AND (NI_LAMP_PICK_8 OR ((NI_FAULT_MUCH_LAMP_PICK_8 OR NI_FAULT_FALSE_LAMP_PICK_8) AND Get100msClk()));
LAMP_PICK_9 := P_On AND (NI_LAMP_PICK_9 OR ((NI_FAULT_MUCH_LAMP_PICK_9 OR NI_FAULT_FALSE_LAMP_PICK_9) AND Get100msClk()));
LAMP_PICK_10 := P_On AND (NI_LAMP_PICK_10 OR ((NI_FAULT_MUCH_LAMP_PICK_10 OR NI_FAULT_FALSE_LAMP_PICK_10) AND Get100msClk()));
LAMP_PICK_11 := P_On AND (NI_LAMP_PICK_11 OR ((NI_FAULT_MUCH_LAMP_PICK_11 OR NI_FAULT_FALSE_LAMP_PICK_11) AND Get100msClk()));
LAMP_PICK_12 := P_On AND (NI_LAMP_PICK_12 OR ((NI_FAULT_MUCH_LAMP_PICK_12 OR NI_FAULT_FALSE_LAMP_PICK_12) AND Get100msClk()));
LAMP_PICK_13 := P_On AND (NI_LAMP_PICK_13 OR ((NI_FAULT_MUCH_LAMP_PICK_13 OR NI_FAULT_FALSE_LAMP_PICK_13) AND Get100msClk()));
LAMP_PICK_14 := P_On AND (NI_LAMP_PICK_14 OR ((NI_FAULT_MUCH_LAMP_PICK_14 OR NI_FAULT_FALSE_LAMP_PICK_14) AND Get100msClk()));
LAMP_PICK_15 := P_On AND (NI_LAMP_PICK_15 OR ((NI_FAULT_MUCH_LAMP_PICK_15 OR NI_FAULT_FALSE_LAMP_PICK_15) AND Get100msClk()));
LAMP_PICK_16 := P_On AND (NI_LAMP_PICK_16 OR ((NI_FAULT_MUCH_LAMP_PICK_16 OR NI_FAULT_FALSE_LAMP_PICK_16) AND Get100msClk()));
LAMP_PICK_17 := P_On AND (NI_LAMP_PICK_17 OR ((NI_FAULT_MUCH_LAMP_PICK_17 OR NI_FAULT_FALSE_LAMP_PICK_17) AND Get100msClk()));
LAMP_PICK_18 := P_On AND (NI_LAMP_PICK_18 OR ((NI_FAULT_MUCH_LAMP_PICK_18 OR NI_FAULT_FALSE_LAMP_PICK_18) AND Get100msClk()));
LAMP_PICK_19 := P_On AND (NI_LAMP_PICK_19 OR ((NI_FAULT_MUCH_LAMP_PICK_19 OR NI_FAULT_FALSE_LAMP_PICK_19) AND Get100msClk()));
LAMP_PICK_20 := P_On AND (NI_LAMP_PICK_20 OR ((NI_FAULT_MUCH_LAMP_PICK_20 OR NI_FAULT_FALSE_LAMP_PICK_20) AND Get100msClk()));

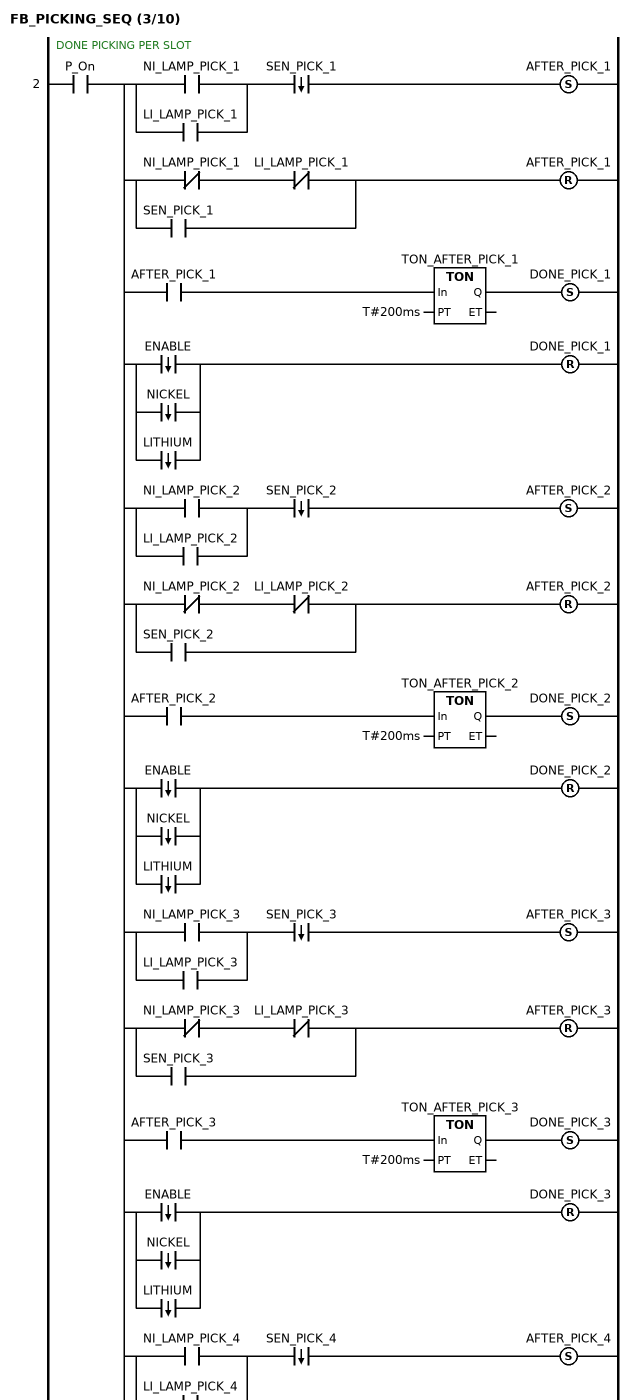

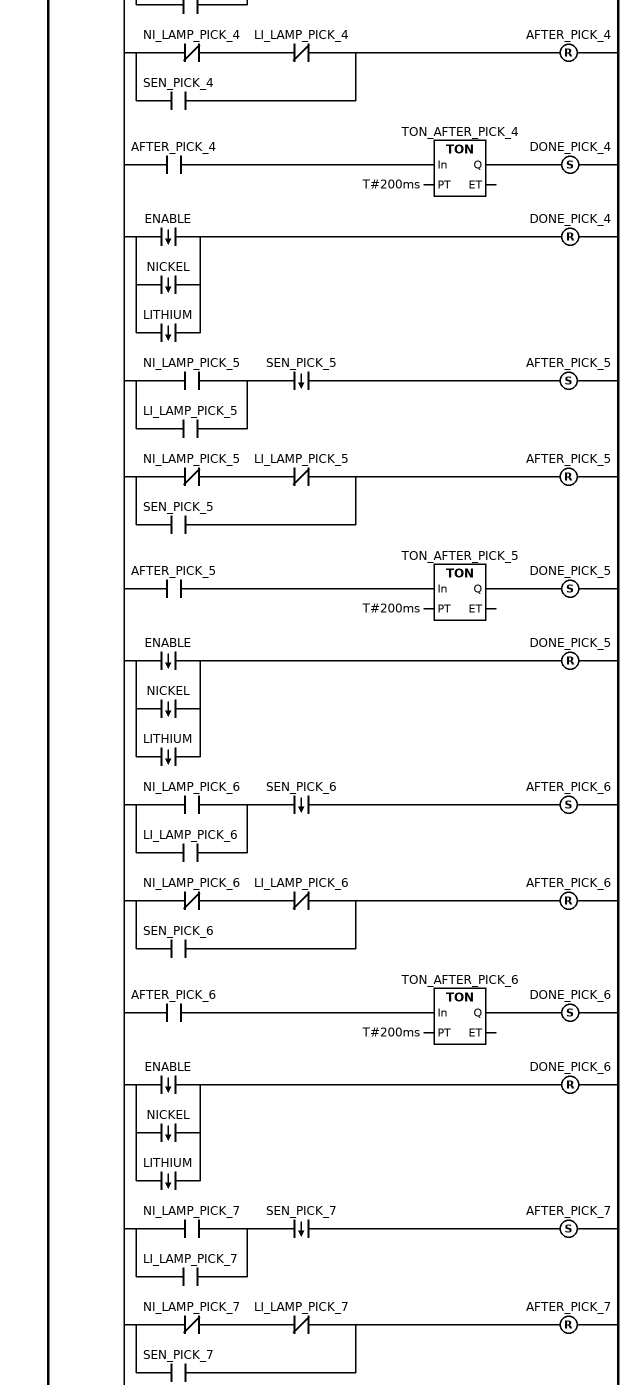

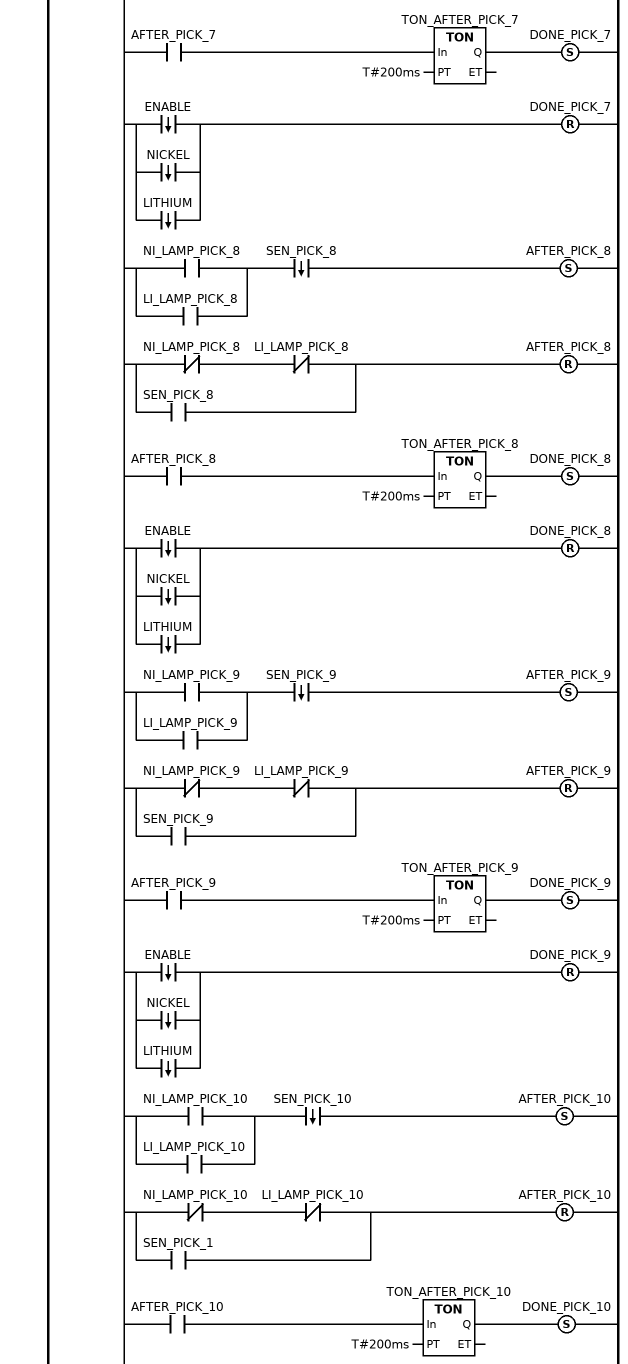

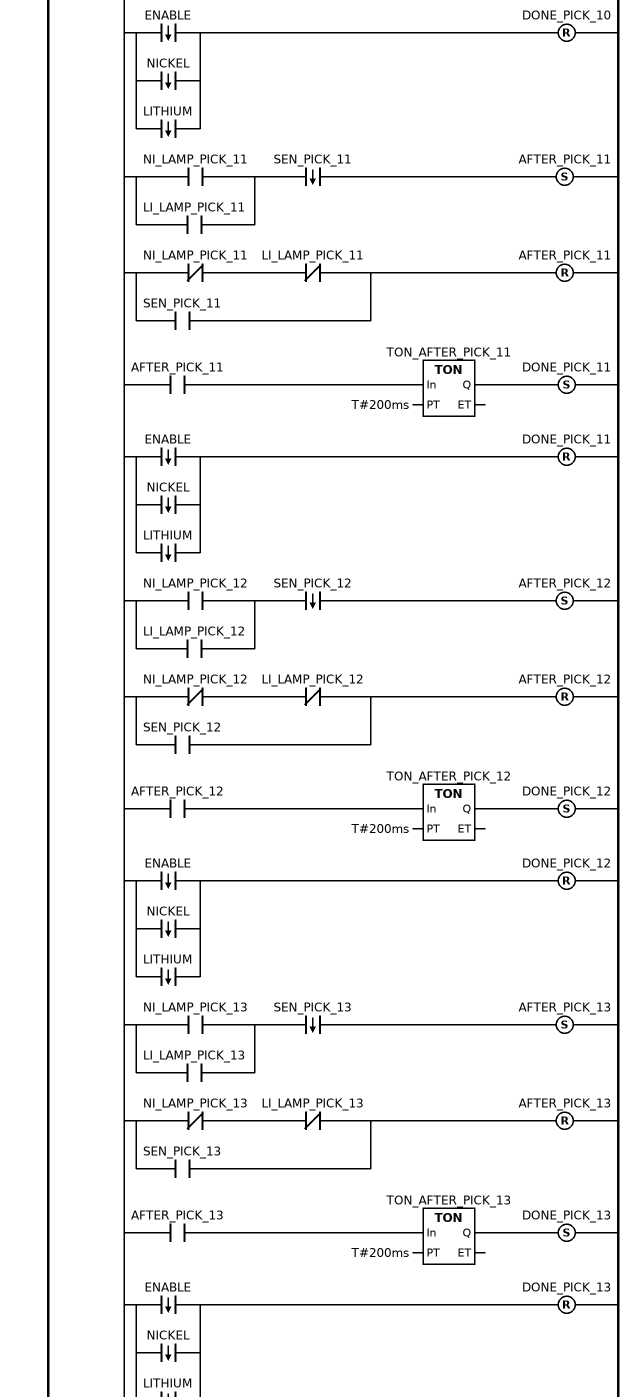

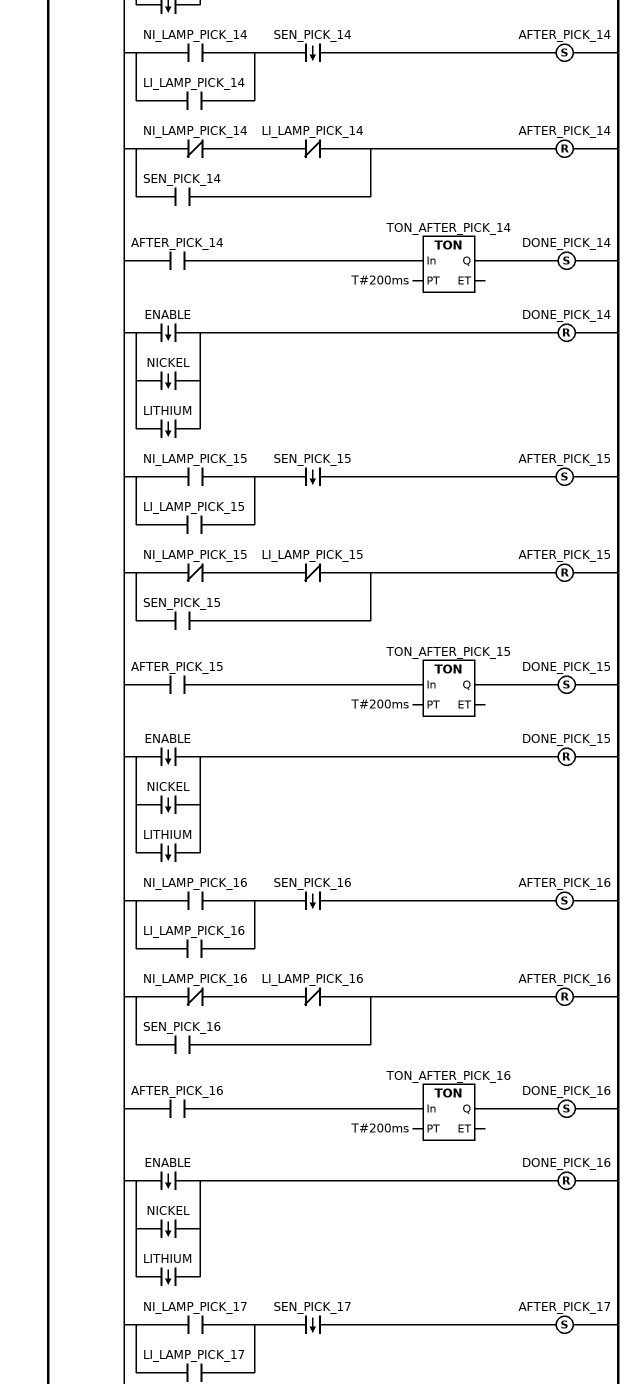

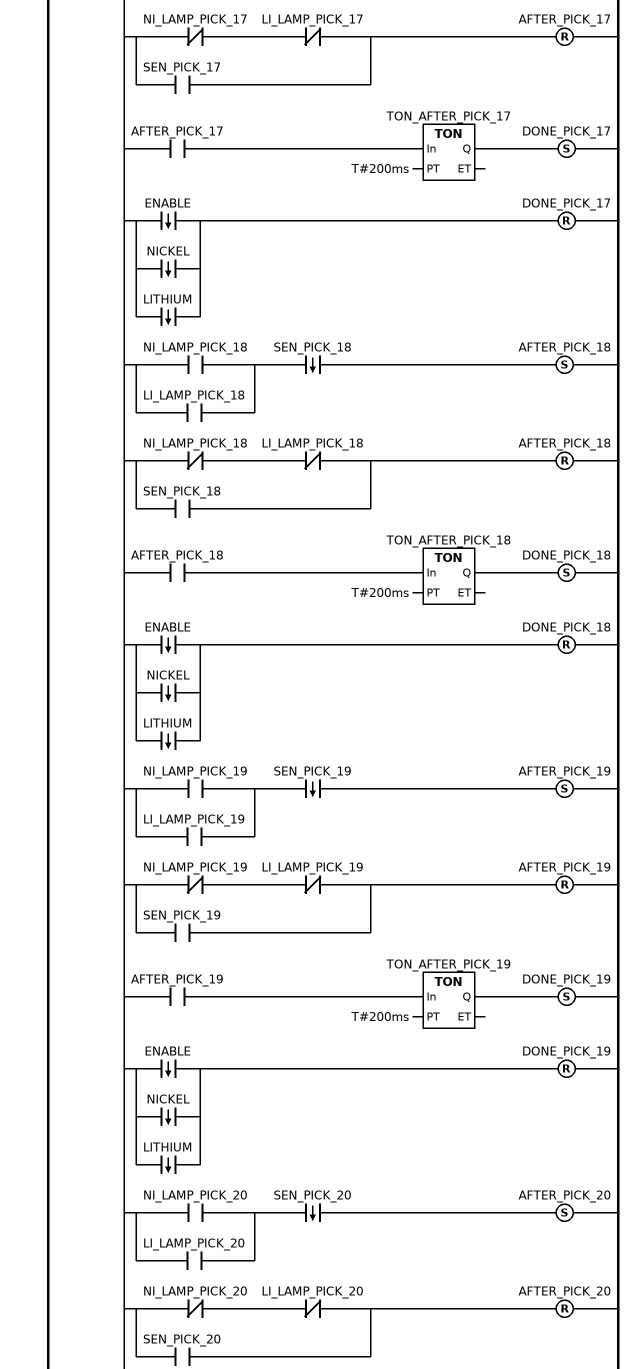

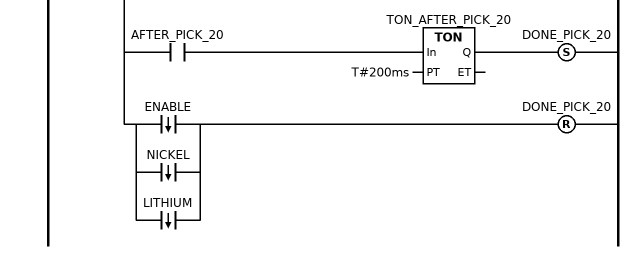
(* Rung 2: DONE PICKING PER SLOT *)
_e12(CLK := SEN_PICK_1);
IF P_On AND (NI_LAMP_PICK_1 OR LI_LAMP_PICK_1) AND _e12.Q THEN AFTER_PICK_1 := TRUE; END_IF;
IF P_On AND ((NOT NI_LAMP_PICK_1 AND NOT LI_LAMP_PICK_1) OR SEN_PICK_1) THEN
    AFTER_PICK_1 := FALSE;
END_IF;
TON_AFTER_PICK_1(In := P_On AND AFTER_PICK_1, PT := T#200ms);
IF TON_AFTER_PICK_1.Q THEN DONE_PICK_1 := TRUE; END_IF;
_e13(CLK := ENABLE);
_e14(CLK := NICKEL);
_e15(CLK := LITHIUM);
IF P_On AND (_e13.Q OR _e14.Q OR _e15.Q) THEN DONE_PICK_1 := FALSE; END_IF;
_e16(CLK := SEN_PICK_2);
IF P_On AND (NI_LAMP_PICK_2 OR LI_LAMP_PICK_2) AND _e16.Q THEN AFTER_PICK_2 := TRUE; END_IF;
IF P_On AND ((NOT NI_LAMP_PICK_2 AND NOT LI_LAMP_PICK_2) OR SEN_PICK_2) THEN
    AFTER_PICK_2 := FALSE;
END_IF;
TON_AFTER_PICK_2(In := P_On AND AFTER_PICK_2, PT := T#200ms);
IF TON_AFTER_PICK_2.Q THEN DONE_PICK_2 := TRUE; END_IF;
_e17(CLK := ENABLE);
_e18(CLK := NICKEL);
_e19(CLK := LITHIUM);
IF P_On AND (_e17.Q OR _e18.Q OR _e19.Q) THEN DONE_PICK_2 := FALSE; END_IF;
_e20(CLK := SEN_PICK_3);
IF P_On AND (NI_LAMP_PICK_3 OR LI_LAMP_PICK_3) AND _e20.Q THEN AFTER_PICK_3 := TRUE; END_IF;
IF P_On AND ((NOT NI_LAMP_PICK_3 AND NOT LI_LAMP_PICK_3) OR SEN_PICK_3) THEN
    AFTER_PICK_3 := FALSE;
END_IF;
TON_AFTER_PICK_3(In := P_On AND AFTER_PICK_3, PT := T#200ms);
IF TON_AFTER_PICK_3.Q THEN DONE_PICK_3 := TRUE; END_IF;
_e21(CLK := ENABLE);
_e22(CLK := NICKEL);
_e23(CLK := LITHIUM);
IF P_On AND (_e21.Q OR _e22.Q OR _e23.Q) THEN DONE_PICK_3 := FALSE; END_IF;
_e24(CLK := SEN_PICK_4);
IF P_On AND (NI_LAMP_PICK_4 OR LI_LAMP_PICK_4) AND _e24.Q THEN AFTER_PICK_4 := TRUE; END_IF;
IF P_On AND ((NOT NI_LAMP_PICK_4 AND NOT LI_LAMP_PICK_4) OR SEN_PICK_4) THEN
    AFTER_PICK_4 := FALSE;
END_IF;
TON_AFTER_PICK_4(In := P_On AND AFTER_PICK_4, PT := T#200ms);
IF TON_AFTER_PICK_4.Q THEN DONE_PICK_4 := TRUE; END_IF;
_e25(CLK := ENABLE);
_e26(CLK := NICKEL);
_e27(CLK := LITHIUM);
IF P_On AND (_e25.Q OR _e26.Q OR _e27.Q) THEN DONE_PICK_4 := FALSE; END_IF;
_e28(CLK := SEN_PICK_5);
IF P_On AND (NI_LAMP_PICK_5 OR LI_LAMP_PICK_5) AND _e28.Q THEN AFTER_PICK_5 := TRUE; END_IF;
IF P_On AND ((NOT NI_LAMP_PICK_5 AND NOT LI_LAMP_PICK_5) OR SEN_PICK_5) THEN
    AFTER_PICK_5 := FALSE;
END_IF;
TON_AFTER_PICK_5(In := P_On AND AFTER_PICK_5, PT := T#200ms);
IF TON_AFTER_PICK_5.Q THEN DONE_PICK_5 := TRUE; END_IF;
_e29(CLK := ENABLE);
_e30(CLK := NICKEL);
_e31(CLK := LITHIUM);
IF P_On AND (_e29.Q OR _e30.Q OR _e31.Q) THEN DONE_PICK_5 := FALSE; END_IF;
_e32(CLK := SEN_PICK_6);
IF P_On AND (NI_LAMP_PICK_6 OR LI_LAMP_PICK_6) AND _e32.Q THEN AFTER_PICK_6 := TRUE; END_IF;
IF P_On AND ((NOT NI_LAMP_PICK_6 AND NOT LI_LAMP_PICK_6) OR SEN_PICK_6) THEN
    AFTER_PICK_6 := FALSE;
END_IF;
TON_AFTER_PICK_6(In := P_On AND AFTER_PICK_6, PT := T#200ms);
IF TON_AFTER_PICK_6.Q THEN DONE_PICK_6 := TRUE; END_IF;
_e33(CLK := ENABLE);
_e34(CLK := NICKEL);
_e35(CLK := LITHIUM);
IF P_On AND (_e33.Q OR _e34.Q OR _e35.Q) THEN DONE_PICK_6 := FALSE; END_IF;
_e36(CLK := SEN_PICK_7);
IF P_On AND (NI_LAMP_PICK_7 OR LI_LAMP_PICK_7) AND _e36.Q THEN AFTER_PICK_7 := TRUE; END_IF;
IF P_On AND ((NOT NI_LAMP_PICK_7 AND NOT LI_LAMP_PICK_7) OR SEN_PICK_7) THEN
    AFTER_PICK_7 := FALSE;
END_IF;
TON_AFTER_PICK_7(In := P_On AND AFTER_PICK_7, PT := T#200ms);
IF TON_AFTER_PICK_7.Q THEN DONE_PICK_7 := TRUE; END_IF;
_e37(CLK := ENABLE);
_e38(CLK := NICKEL);
_e39(CLK := LITHIUM);
IF P_On AND (_e37.Q OR _e38.Q OR _e39.Q) THEN DONE_PICK_7 := FALSE; END_IF;
_e40(CLK := SEN_PICK_8);
IF P_On AND (NI_LAMP_PICK_8 OR LI_LAMP_PICK_8) AND _e40.Q THEN AFTER_PICK_8 := TRUE; END_IF;
IF P_On AND ((NOT NI_LAMP_PICK_8 AND NOT LI_LAMP_PICK_8) OR SEN_PICK_8) THEN
    AFTER_PICK_8 := FALSE;
END_IF;
TON_AFTER_PICK_8(In := P_On AND AFTER_PICK_8, PT := T#200ms);
IF TON_AFTER_PICK_8.Q THEN DONE_PICK_8 := TRUE; END_IF;
_e41(CLK := ENABLE);
_e42(CLK := NICKEL);
_e43(CLK := LITHIUM);
IF P_On AND (_e41.Q OR _e42.Q OR _e43.Q) THEN DONE_PICK_8 := FALSE; END_IF;
_e44(CLK := SEN_PICK_9);
IF P_On AND (NI_LAMP_PICK_9 OR LI_LAMP_PICK_9) AND _e44.Q THEN AFTER_PICK_9 := TRUE; END_IF;
IF P_On AND ((NOT NI_LAMP_PICK_9 AND NOT LI_LAMP_PICK_9) OR SEN_PICK_9) THEN
    AFTER_PICK_9 := FALSE;
END_IF;
TON_AFTER_PICK_9(In := P_On AND AFTER_PICK_9, PT := T#200ms);
IF TON_AFTER_PICK_9.Q THEN DONE_PICK_9 := TRUE; END_IF;
_e45(CLK := ENABLE);
_e46(CLK := NICKEL);
_e47(CLK := LITHIUM);
IF P_On AND (_e45.Q OR _e46.Q OR _e47.Q) THEN DONE_PICK_9 := FALSE; END_IF;
_e48(CLK := SEN_PICK_10);
IF P_On AND (NI_LAMP_PICK_10 OR LI_LAMP_PICK_10) AND _e48.Q THEN AFTER_PICK_10 := TRUE; END_IF;
IF P_On AND ((NOT NI_LAMP_PICK_10 AND NOT LI_LAMP_PICK_10) OR SEN_PICK_1) THEN
    AFTER_PICK_10 := FALSE;
END_IF;
TON_AFTER_PICK_10(In := P_On AND AFTER_PICK_10, PT := T#200ms);
IF TON_AFTER_PICK_10.Q THEN DONE_PICK_10 := TRUE; END_IF;
_e49(CLK := ENABLE);
_e50(CLK := NICKEL);
_e51(CLK := LITHIUM);
IF P_On AND (_e49.Q OR _e50.Q OR _e51.Q) THEN DONE_PICK_10 := FALSE; END_IF;
_e52(CLK := SEN_PICK_11);
IF P_On AND (NI_LAMP_PICK_11 OR LI_LAMP_PICK_11) AND _e52.Q THEN AFTER_PICK_11 := TRUE; END_IF;
IF P_On AND ((NOT NI_LAMP_PICK_11 AND NOT LI_LAMP_PICK_11) OR SEN_PICK_11) THEN
    AFTER_PICK_11 := FALSE;
END_IF;
TON_AFTER_PICK_11(In := P_On AND AFTER_PICK_11, PT := T#200ms);
IF TON_AFTER_PICK_11.Q THEN DONE_PICK_11 := TRUE; END_IF;
_e53(CLK := ENABLE);
_e54(CLK := NICKEL);
_e55(CLK := LITHIUM);
IF P_On AND (_e53.Q OR _e54.Q OR _e55.Q) THEN DONE_PICK_11 := FALSE; END_IF;
_e56(CLK := SEN_PICK_12);
IF P_On AND (NI_LAMP_PICK_12 OR LI_LAMP_PICK_12) AND _e56.Q THEN AFTER_PICK_12 := TRUE; END_IF;
IF P_On AND ((NOT NI_LAMP_PICK_12 AND NOT LI_LAMP_PICK_12) OR SEN_PICK_12) THEN
    AFTER_PICK_12 := FALSE;
END_IF;
TON_AFTER_PICK_12(In := P_On AND AFTER_PICK_12, PT := T#200ms);
IF TON_AFTER_PICK_12.Q THEN DONE_PICK_12 := TRUE; END_IF;
_e57(CLK := ENABLE);
_e58(CLK := NICKEL);
_e59(CLK := LITHIUM);
IF P_On AND (_e57.Q OR _e58.Q OR _e59.Q) THEN DONE_PICK_12 := FALSE; END_IF;
_e60(CLK := SEN_PICK_13);
IF P_On AND (NI_LAMP_PICK_13 OR LI_LAMP_PICK_13) AND _e60.Q THEN AFTER_PICK_13 := TRUE; END_IF;
IF P_On AND ((NOT NI_LAMP_PICK_13 AND NOT LI_LAMP_PICK_13) OR SEN_PICK_13) THEN
    AFTER_PICK_13 := FALSE;
END_IF;
TON_AFTER_PICK_13(In := P_On AND AFTER_PICK_13, PT := T#200ms);
IF TON_AFTER_PICK_13.Q THEN DONE_PICK_13 := TRUE; END_IF;
_e61(CLK := ENABLE);
_e62(CLK := NICKEL);
_e63(CLK := LITHIUM);
IF P_On AND (_e61.Q OR _e62.Q OR _e63.Q) THEN DONE_PICK_13 := FALSE; END_IF;
_e64(CLK := SEN_PICK_14);
IF P_On AND (NI_LAMP_PICK_14 OR LI_LAMP_PICK_14) AND _e64.Q THEN AFTER_PICK_14 := TRUE; END_IF;
IF P_On AND ((NOT NI_LAMP_PICK_14 AND NOT LI_LAMP_PICK_14) OR SEN_PICK_14) THEN
    AFTER_PICK_14 := FALSE;
END_IF;
TON_AFTER_PICK_14(In := P_On AND AFTER_PICK_14, PT := T#200ms);
IF TON_AFTER_PICK_14.Q THEN DONE_PICK_14 := TRUE; END_IF;
_e65(CLK := ENABLE);
_e66(CLK := NICKEL);
_e67(CLK := LITHIUM);
IF P_On AND (_e65.Q OR _e66.Q OR _e67.Q) THEN DONE_PICK_14 := FALSE; END_IF;
_e68(CLK := SEN_PICK_15);
IF P_On AND (NI_LAMP_PICK_15 OR LI_LAMP_PICK_15) AND _e68.Q THEN AFTER_PICK_15 := TRUE; END_IF;
IF P_On AND ((NOT NI_LAMP_PICK_15 AND NOT LI_LAMP_PICK_15) OR SEN_PICK_15) THEN
    AFTER_PICK_15 := FALSE;
END_IF;
TON_AFTER_PICK_15(In := P_On AND AFTER_PICK_15, PT := T#200ms);
IF TON_AFTER_PICK_15.Q THEN DONE_PICK_15 := TRUE; END_IF;
_e69(CLK := ENABLE);
_e70(CLK := NICKEL);
_e71(CLK := LITHIUM);
IF P_On AND (_e69.Q OR _e70.Q OR _e71.Q) THEN DONE_PICK_15 := FALSE; END_IF;
_e72(CLK := SEN_PICK_16);
IF P_On AND (NI_LAMP_PICK_16 OR LI_LAMP_PICK_16) AND _e72.Q THEN AFTER_PICK_16 := TRUE; END_IF;
IF P_On AND ((NOT NI_LAMP_PICK_16 AND NOT LI_LAMP_PICK_16) OR SEN_PICK_16) THEN
    AFTER_PICK_16 := FALSE;
END_IF;
TON_AFTER_PICK_16(In := P_On AND AFTER_PICK_16, PT := T#200ms);
IF TON_AFTER_PICK_16.Q THEN DONE_PICK_16 := TRUE; END_IF;
_e73(CLK := ENABLE);
_e74(CLK := NICKEL);
_e75(CLK := LITHIUM);
IF P_On AND (_e73.Q OR _e74.Q OR _e75.Q) THEN DONE_PICK_16 := FALSE; END_IF;
_e76(CLK := SEN_PICK_17);
IF P_On AND (NI_LAMP_PICK_17 OR LI_LAMP_PICK_17) AND _e76.Q THEN AFTER_PICK_17 := TRUE; END_IF;
IF P_On AND ((NOT NI_LAMP_PICK_17 AND NOT LI_LAMP_PICK_17) OR SEN_PICK_17) THEN
    AFTER_PICK_17 := FALSE;
END_IF;
TON_AFTER_PICK_17(In := P_On AND AFTER_PICK_17, PT := T#200ms);
IF TON_AFTER_PICK_17.Q THEN DONE_PICK_17 := TRUE; END_IF;
_e77(CLK := ENABLE);
_e78(CLK := NICKEL);
_e79(CLK := LITHIUM);
IF P_On AND (_e77.Q OR _e78.Q OR _e79.Q) THEN DONE_PICK_17 := FALSE; END_IF;
_e80(CLK := SEN_PICK_18);
IF P_On AND (NI_LAMP_PICK_18 OR LI_LAMP_PICK_18) AND _e80.Q THEN AFTER_PICK_18 := TRUE; END_IF;
IF P_On AND ((NOT NI_LAMP_PICK_18 AND NOT LI_LAMP_PICK_18) OR SEN_PICK_18) THEN
    AFTER_PICK_18 := FALSE;
END_IF;
TON_AFTER_PICK_18(In := P_On AND AFTER_PICK_18, PT := T#200ms);
IF TON_AFTER_PICK_18.Q THEN DONE_PICK_18 := TRUE; END_IF;
_e81(CLK := ENABLE);
_e82(CLK := NICKEL);
_e83(CLK := LITHIUM);
IF P_On AND (_e81.Q OR _e82.Q OR _e83.Q) THEN DONE_PICK_18 := FALSE; END_IF;
_e84(CLK := SEN_PICK_19);
IF P_On AND (NI_LAMP_PICK_19 OR LI_LAMP_PICK_19) AND _e84.Q THEN AFTER_PICK_19 := TRUE; END_IF;
IF P_On AND ((NOT NI_LAMP_PICK_19 AND NOT LI_LAMP_PICK_19) OR SEN_PICK_19) THEN
    AFTER_PICK_19 := FALSE;
END_IF;
TON_AFTER_PICK_19(In := P_On AND AFTER_PICK_19, PT := T#200ms);
IF TON_AFTER_PICK_19.Q THEN DONE_PICK_19 := TRUE; END_IF;
_e85(CLK := ENABLE);
_e86(CLK := NICKEL);
_e87(CLK := LITHIUM);
IF P_On AND (_e85.Q OR _e86.Q OR _e87.Q) THEN DONE_PICK_19 := FALSE; END_IF;
_e88(CLK := SEN_PICK_20);
IF P_On AND (NI_LAMP_PICK_20 OR LI_LAMP_PICK_20) AND _e88.Q THEN AFTER_PICK_20 := TRUE; END_IF;
IF P_On AND ((NOT NI_LAMP_PICK_20 AND NOT LI_LAMP_PICK_20) OR SEN_PICK_20) THEN
    AFTER_PICK_20 := FALSE;
END_IF;
TON_AFTER_PICK_20(In := P_On AND AFTER_PICK_20, PT := T#200ms);
IF TON_AFTER_PICK_20.Q THEN DONE_PICK_20 := TRUE; END_IF;
_e89(CLK := ENABLE);
_e90(CLK := NICKEL);
_e91(CLK := LITHIUM);
IF P_On AND (_e89.Q OR _e90.Q OR _e91.Q) THEN DONE_PICK_20 := FALSE; END_IF;

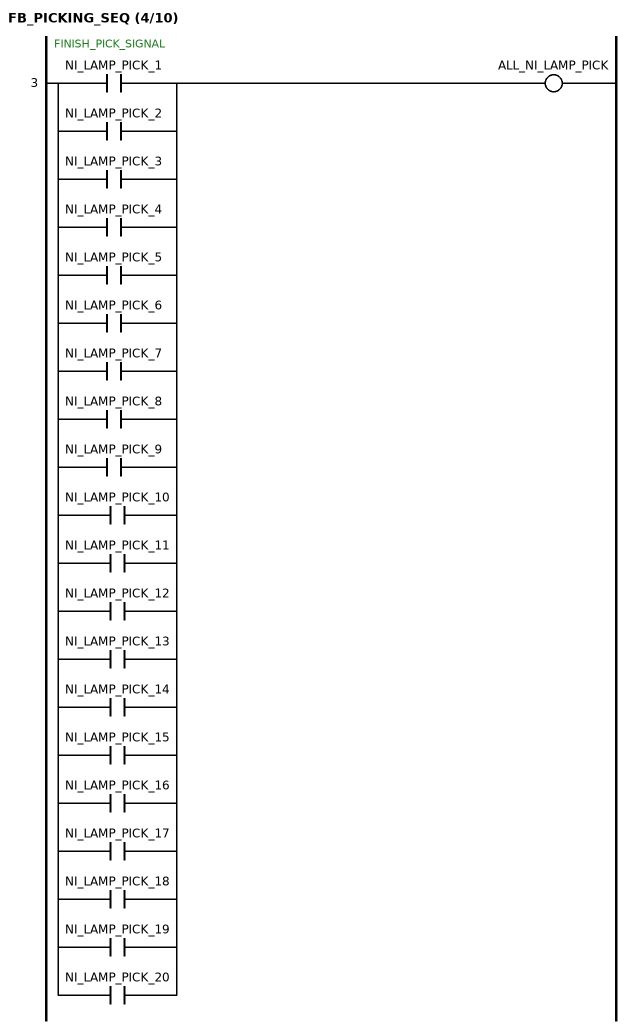
(* Rung 3: FINISH_PICK_SIGNAL *)
ALL_NI_LAMP_PICK := NI_LAMP_PICK_1 OR NI_LAMP_PICK_2 OR NI_LAMP_PICK_3 OR NI_LAMP_PICK_4 OR NI_LAMP_PICK_5 OR NI_LAMP_PICK_6 OR NI_LAMP_PICK_7 OR NI_LAMP_PICK_8 OR NI_LAMP_PICK_9 OR NI_LAMP_PICK_10 OR NI_LAMP_PICK_11 OR NI_LAMP_PICK_12 OR NI_LAMP_PICK_13 OR NI_LAMP_PICK_14 OR NI_LAMP_PICK_15 OR NI_LAMP_PICK_16 OR NI_LAMP_PICK_17 OR NI_LAMP_PICK_18 OR NI_LAMP_PICK_19 OR NI_LAMP_PICK_20;

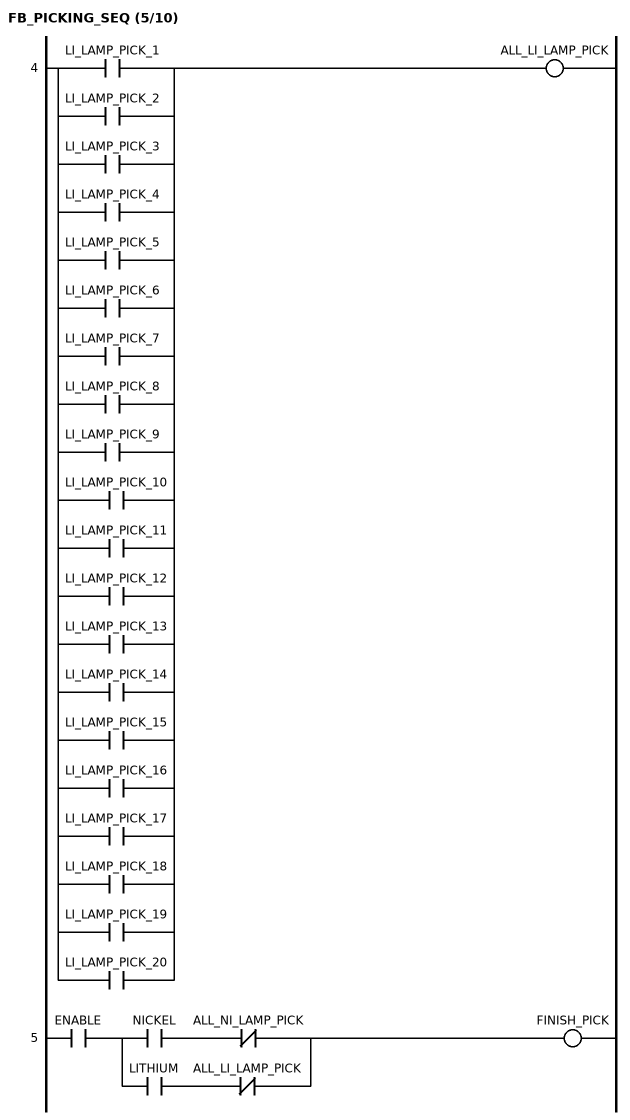
(* Rung 4 *)
ALL_LI_LAMP_PICK := LI_LAMP_PICK_1 OR LI_LAMP_PICK_2 OR LI_LAMP_PICK_3 OR LI_LAMP_PICK_4 OR LI_LAMP_PICK_5 OR LI_LAMP_PICK_6 OR LI_LAMP_PICK_7 OR LI_LAMP_PICK_8 OR LI_LAMP_PICK_9 OR LI_LAMP_PICK_10 OR LI_LAMP_PICK_11 OR LI_LAMP_PICK_12 OR LI_LAMP_PICK_13 OR LI_LAMP_PICK_14 OR LI_LAMP_PICK_15 OR LI_LAMP_PICK_16 OR LI_LAMP_PICK_17 OR LI_LAMP_PICK_18 OR LI_LAMP_PICK_19 OR LI_LAMP_PICK_20;
(* Rung 5 *)
FINISH_PICK := ENABLE AND ((NICKEL AND NOT ALL_NI_LAMP_PICK) OR (LITHIUM AND NOT ALL_LI_LAMP_PICK));

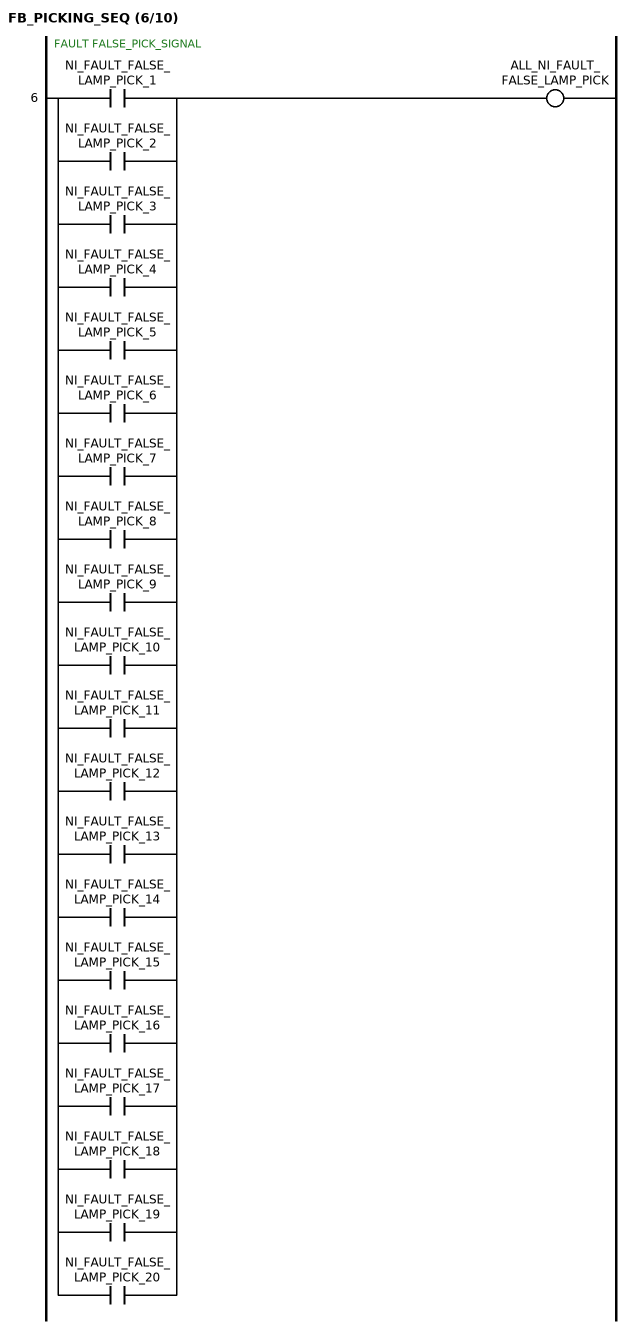
(* Rung 6: FAULT FALSE_PICK_SIGNAL *)
ALL_NI_FAULT_FALSE_LAMP_PICK := NI_FAULT_FALSE_LAMP_PICK_1 OR NI_FAULT_FALSE_LAMP_PICK_2 OR NI_FAULT_FALSE_LAMP_PICK_3 OR NI_FAULT_FALSE_LAMP_PICK_4 OR NI_FAULT_FALSE_LAMP_PICK_5 OR NI_FAULT_FALSE_LAMP_PICK_6 OR NI_FAULT_FALSE_LAMP_PICK_7 OR NI_FAULT_FALSE_LAMP_PICK_8 OR NI_FAULT_FALSE_LAMP_PICK_9 OR NI_FAULT_FALSE_LAMP_PICK_10 OR NI_FAULT_FALSE_LAMP_PICK_11 OR NI_FAULT_FALSE_LAMP_PICK_12 OR NI_FAULT_FALSE_LAMP_PICK_13 OR NI_FAULT_FALSE_LAMP_PICK_14 OR NI_FAULT_FALSE_LAMP_PICK_15 OR NI_FAULT_FALSE_LAMP_PICK_16 OR NI_FAULT_FALSE_LAMP_PICK_17 OR NI_FAULT_FALSE_LAMP_PICK_18 OR NI_FAULT_FALSE_LAMP_PICK_19 OR NI_FAULT_FALSE_LAMP_PICK_20;

